ABB RAPID module: 3RHTCO_Mod1(Mod)_5000.mod

MODULE RHTCO1
    ! Code Developers: Linus Y L Ang and Zhang Zhiqian (IHPC/EM)
    ! Version Date/Time: 2024.12.02 / 16:41

    ! Get input coordinates.
    PERS num x_coords_rel{5000}:=[0.0, 0.2, 0.0, 0.1, 0.0, 0.2, 0.0, 0.1, 0.0, 0.2, 0.0, 0.0, -0.2, 0.0, -0.1, 0.0, 0.0, -0.2, 0.0, -0.1, 0.0, 0.0, -0.2, 0.0, -0.2, 0.0, 0.0, -0.1, 0.0, -0.2, 0.0, -0.1, -4.9, 0.0, 5.0, 0.0, 0.2, 0.0, 0.1, 0.0, 0.2, 0.0, 0.2, 0.0, 0.1, 0.0, 0.2, 0.0, 0.1, 0.0, 0.2, 0.0, 0.0, 0.0, -0.2, 0.0, -0.1, 0.0, -0.2, 0.0, -0.1, 0.0, 0.0, -0.2, 0.0, -0.2, 0.0, -0.1, 0.0, -0.2, 0.0, 0.0, -0.1, -4.9, 0.0, 4.9, 0.0, 0.1, 0.0, 0.2, 0.0, 0.1, 0.0, 0.2, 0.0, 0.2, 0.0, 0.1, 0.0, 0.2, 0.0, 0.1, 0.0, 0.2, 0.0, 0.0, -0.2, 0.0, -0.1, 0.0, -0.2, 0.0, -0.1, 0.0, 0.0, -0.2, 0.0, -0.2, 0.0, -0.1, 0.0, -0.2, 0.0, -0.1, -0.2, -4.7, 0.0, 4.7, 0.0, 0.2, 0.1, 0.0, 0.2, 0.1, 0.0, 0.2, 0.0, 0.2, 0.0, 0.1, 0.0, 0.2, 0.0, 0.1, 0.0, 0.2, 0.0, 0.2, -0.2, 0.0, -0.2, 0.0, -0.1, 0.0, 0.0, -0.2, 0.0, -0.1, 0.0, -0.2, 0.0, -0.2, 0.0, -0.1, 0.0, -0.2, 0.0, -0.1, -4.9, 0.0, 4.9, 0.0, 0.1, 0.2, 0.0, 0.0, 0.1, 0.0, 0.2, 0.0, 0.2, 0.0, 0.1, 0.0, 0.2, 0.0, 0.1, 0.0, 0.2, 0.0, 0.2, 0.0, 0.0, -0.2, 0.0, -0.2, 0.0, -0.1, -0.2, 0.0, -0.1, 0.0, -0.2, 0.0, -0.2, 0.0, -0.1, -0.2, 0.0, -0.1, 0.0, -0.2, -0.2, -0.1, -0.2, -0.2, -1.1, -0.1, -1.2, -0.1, -1.1, -0.2, -0.2, 0.0, 0.2, 0.0, 0.2, 1.1, 0.1, 1.2, 0.1, 1.1, 0.2, 0.2, 0.1, 0.2, 0.2, 0.0, 0.0, 0.1, 0.0, 0.2, 0.0, 0.0, 0.1, 0.0, 0.0, 0.2, 0.0, 0.0, 0.2, -0.2, -0.2, -0.1, -0.2, -1.0, -0.1, -1.0, -0.1, -1.2, -0.1, 0.0, 0.1, 1.2, 0.1, 1.0, 0.1, 1.0, 0.2, 0.1, 0.2, 0.2, 0.1, 0.0, 0.2, 0.1, 0.2, 0.2, 0.1, 0.2, 0.1, 0.2, 0.2, 0.1, 0.2, 0.0, -0.2, 0.0, -0.1, 0.0, -0.2, -0.2, -0.1, -0.2, -0.1, -0.2, -0.2, -0.1, -0.2, -0.1, -0.2, 0.0, 0.2, 0.1, 0.2, 0.1, 0.2, 0.2, 0.1, 0.2, 0.1, 0.8, 0.0, 0.2, 0.2, 0.1, 0.2, 0.1, 0.2, 0.2, 0.1, 0.2, 0.2, 0.1, 0.2, 0.1, 0.2, 0.2, 0.1, 0.2, 0.1, 0.0, -0.1, 0.0, -0.2, 0.0, -0.1, 0.0, -0.2, -0.2, -0.1, -0.2, -0.1, -0.2, -0.2, -0.1, -0.2, -0.2, -0.1, -0.2, -0.1, -0.2, -0.2, -0.1, -0.2, -0.1, -0.2, -0.2, -0.1, -0.7, -0.1, -0.7, -0.1, -0.2, -0.1, -0.2, -0.2, -0.8, 0.0, 0.2, 0.0, 0.0, 0.1, 0.0, 0.0, 0.0, 0.2, 0.0, 0.0, 0.2, 0.0, 0.0, 0.1, 0.0, -0.1, 0.0, -0.2, 0.0, 0.0, -0.2, 0.0, 0.0, -0.1, 0.0, 0.0, 0.0, -0.2, 0.0, 0.0, -0.1, 0.0, -0.2, -0.2, -0.1, -0.2, -0.1, -0.2, -0.2, -0.1, -0.2, -0.1, -0.2, -0.2, -0.1, -0.2, -0.1, -0.2, -0.2, -0.1, -0.2, -0.1, -3.27, -0.16, 3.43, -0.2, 0.0, 0.0, 0.0, -0.2, 0.0, 0.0, 0.0, -0.13, 0.0, 0.0, 0.0, -0.16, 0.0, 0.0, -0.16, -0.16, -0.17, -0.16, -0.16, -0.16, -0.16, -0.16, -0.16, -0.16, -0.16, -0.16, -0.16, -0.16, -0.16, -0.17, -0.16, -0.16, -0.16, -0.16, -0.16, -0.16, -0.16, -0.16, -0.16, -0.16, -0.16, -0.16, -0.17, -0.16, -0.16, -0.16, -0.16, -0.16, -0.16, -0.16, -0.16, -0.16, -0.16, -0.16, -0.16, -0.17, -0.16, -0.16, -0.16, -0.16, 0.16, 0.16, 0.16, 0.16, 0.17, 0.16, 0.16, 0.16, 0.16, 0.16, 0.16, 0.16, 0.16, 0.16, 0.16, 0.16, 0.16, 0.17, 0.16, 0.16, 0.16, 0.16, 0.16, 0.16, 0.0, -0.8, -4.34, 0.0, 4.18, 0.0, 0.16, 0.0, 0.0, 0.16, 0.0, 0.16, 0.0, 0.16, 0.0, 0.16, 0.0, 0.16, 0.0, 0.16, 0.0, 0.0, -0.16, -0.16, -0.16, -0.16, -0.16, -0.16, -0.16, -0.17, -0.16, -0.16, -0.16, -0.16, -0.16, -0.16, -0.16, -0.16, 0.0, 0.16, 0.16, 0.16, 0.16, 0.16, 0.16, 0.16, 0.16, 0.17, 0.16, 0.16, 0.16, 0.16, 0.16, 0.16, 0.16, 0.0, -0.16, 0.0, -0.16, 0.0, -0.16, 0.0, -0.16, 0.0, -0.16, 0.0, 0.64, 0.16, 0.0, 0.16, 0.16, 0.16, 0.16, 0.16, 0.17, 0.16, 0.16, 0.16, 0.16, 0.16, 0.16, 0.16, 0.16, 0.16, 0.16, 0.16, 0.16, 0.17, 0.16, 0.16, 0.29, 0.0, 0.0, 0.0, 0.2, 0.0, 0.0, 0.0, 0.2, 0.0, 0.0, 0.0, 0.1, 0.2, 0.1, 0.2, 0.2, 0.1, 0.2, 0.1, 0.2, 0.2, 0.1, 0.2, 0.1, 0.2, 0.2, 0.1, 0.2, 0.1, 0.2, 0.2, 0.0, 0.1, 0.2, 0.6, 0.2, 0.2, 0.1, 0.2, 0.1, 0.7, 0.1, 0.7, 0.1, 0.2, 0.2, 0.1, 0.2, 0.1, 0.0, 0.0, 0.0, -0.1, 0.0, 0.0, -0.2, 0.0, 0.0, -0.1, 0.0, 0.0, -0.2, 0.0, 0.0, 0.0, -0.2, 0.0, 0.0, -0.1, -0.2, -0.1, -0.2, -0.2, -0.1, -0.2, -0.1, -0.2, -0.2, -0.1, -0.2, -0.1, -0.2, -0.2, -0.1, -0.2, -0.2, 0.0, 0.2, 0.2, 0.1, 0.2, 0.2, 0.1, 0.2, 0.1, 0.2, 0.2, 0.1, 0.2, 0.1, 0.2, 0.2, 0.1, 0.2, 0.1, 0.4, 0.0, 0.0, 0.0, 0.1, 0.0, 0.0, 0.2, 0.0, 0.0, 0.1, 0.0, 0.0, 0.2, 0.0, 0.0, 0.2, 0.1, 0.2, 0.1, 0.2, 0.2, 0.1, 0.2, 0.2, 0.1, 0.2, 0.1, 0.2, 0.6, 0.0, 0.2, 0.2, 0.1, 0.2, 0.1, 0.2, 0.2, 0.1, 0.2, 0.1, 0.2, 0.2, 0.1, 0.2, 0.2, 0.1, 0.2, 0.1, 0.2, 0.2, 0.0, 0.0, 0.0, 0.1, 0.0, 0.0, 0.0, 0.2, 0.0, 0.0, 0.0, 0.1, 0.0, 0.0, 0.2, 0.0, 0.0, 0.0, 0.2, 0.0, 0.0, 0.0, 0.1, 0.0, 0.0, 0.0, -0.1, 0.0, -0.2, -0.2, -0.1, -0.2, -0.1, -0.2, -0.2, -0.1, -0.2, -0.1, -0.2, -0.2, -0.1, -0.2, -0.2, -0.1, -0.2, -0.1, -0.2, -0.2, -0.1, -0.2, -0.1, -0.2, 0.0, 0.2, 0.1, 0.2, 0.1, 0.2, 0.2, 0.1, 0.2, 0.1, 0.2, 0.2, 0.1, 0.2, 0.2, 0.1, 0.2, 0.1, 0.2, 0.2, 0.1, 0.2, 0.1, 0.2, 0.0, 0.2, 0.0, 0.1, 0.0, 0.2, 0.0, 0.0, 0.1, 0.0, 0.2, 0.0, 0.0, 0.2, 0.0, 0.1, 0.0, 0.2, 0.0, 0.0, 0.1, 0.0, 0.2, 0.0, 0.2, 0.0, 0.0, -0.2, -0.2, 0.0, -0.1, -0.2, 0.0, -0.1, -0.2, -0.2, 0.0, -0.1, -0.2, 0.0, -0.1, -0.2, 0.0, -0.2, -0.1, -0.2, 0.0, -0.1, -0.2, -0.2, -0.8, -0.1, -0.2, -0.2, 0.0, 0.2, 0.2, 0.1, 1.0, 0.5, 0.0, 0.1, 0.2, 0.2, 0.0, 0.1, 0.2, 0.0, 0.1, 0.2, 0.0, 0.2, 0.1, 0.2, 0.0, 0.1, 0.2, 0.0, 0.2, 0.1, -0.1, -0.2, 0.0, -0.2, 0.0, 0.0, -0.1, 0.0, -0.2, 0.0, -0.1, 0.0, 0.0, -0.2, 0.0, -0.2, 0.0, 0.0, -0.1, 0.0, -0.2, 0.0, -0.1, 0.0, 0.1, 0.0, 0.2, 0.1, 0.2, 0.2, 0.1, 0.2, 0.6, 0.2, 0.1, 0.2, 0.2, 0.1, 0.2, 0.2, 0.1, 0.2, 0.6, 0.2, 0.1, 0.2, 0.2, 0.1, 0.2, 0.1, 0.2, 0.2, 0.6, 0.0, -0.6, -0.2, -0.2, -0.1, -0.2, -0.1, -0.2, -0.2, -0.1, -0.2, -0.6, -0.2, -0.1, -0.2, -0.2, -0.1, -0.2, -0.2, -0.1, -0.2, -0.6, -0.2, -0.1, -0.2, -0.2, -0.1, -0.2, 0.0, 0.0, 0.0, -0.1, 0.0, 0.0, 0.0, -0.2, 0.0, 0.0, -0.2, 0.0, 0.0, 0.0, -0.1, 0.0, 0.0, 0.0, -0.2, 0.0, 0.0, 0.0, -0.1, 0.0, 0.8, 0.1, 1.1, 0.2, 1.0, 0.1, 0.0, -0.1, -1.0, -0.2, -1.1, -0.1, -0.8, -0.2, -0.2, -0.1, -0.2, -0.1, -0.2, -0.2, -0.1, -0.2, -0.2, -0.1, -0.2, -0.1, -0.2, -0.2, -0.1, -0.2, -0.1, -0.2, -0.2, -0.1, -0.2, 0.0, 0.2, 0.0, 0.1, 0.0, 0.2, 0.0, 0.0, 0.2, 0.1, 0.2, 0.1, 0.2, 0.2, 0.0, -0.2, -0.2, -0.1, -0.2, -0.1, -0.2, -0.2, -0.1, -0.2, -0.1, -0.2, -0.2, -0.1, -0.2, -0.1, -0.2, -0.2, -0.1, -0.2, -0.2, -0.1, -0.2, -0.1, -0.2, -0.2, -0.1, -0.2, 0.0, 0.2, 0.0, 0.1, 0.0, 0.2, 0.2, 0.1, 0.2, 0.8, 0.2, 0.8, 0.1, 0.8, 0.2, 0.0, -0.2, -0.8, -0.1, -0.8, -0.2, -0.8, -0.2, -0.6, -0.2, -0.1, -0.2, -0.2, -0.1, -0.2, -0.1, -0.2, -0.2, -0.1, -0.2, -0.1, 0.0, 0.0, -0.2, 0.0, 0.0, -0.2, 0.0, 0.0, -0.1, 0.0, -0.2, 0.0, 0.0, -0.1, 0.0, 0.0, 0.1, 0.0, 0.2, 0.0, 0.1, 0.2, 0.0, 0.2, 0.0, 0.1, 0.0, 0.2, 0.0, 0.1, 0.2, 0.0, 0.2, 0.0, 0.1, 4.7, 0.0, -4.5, -0.2, -0.1, 0.0, -0.2, 0.0, -0.2, 0.0, -0.1, 0.0, -0.2, 0.0, -0.1, 0.0, -0.2, 0.0, -0.2, 0.0, 0.0, -0.1, 0.0, -0.2, 0.2, 0.0, 0.1, 0.0, 0.2, 0.0, 0.2, 0.0, 0.1, 0.0, 0.2, 0.0, 0.1, 0.0, 0.0, 0.2, 0.0, 0.2, 0.1, 4.5, 0.0, -4.5, -0.1, 0.0, -0.2, 0.0, -0.2, 0.0, -0.1, 0.0, -0.2, 0.0, -0.1, 0.0, -0.2, 0.0, -0.2, -0.1, 0.0, -0.2, 0.0, 0.0, 0.0, 0.2, 0.0, 0.1, 0.0, 0.2, 0.0, 0.2, 0.0, 0.1, 0.0, 0.0, 0.2, 0.0, 0.1, 0.0, 0.2, 0.0, 0.2, 0.1, 4.7, 0.0, -4.8, -0.2, 0.0, -0.2, 0.0, -0.1, 0.0, -0.2, 0.0, -0.1, 0.0, -0.2, 0.0, -0.2, 0.0, -0.1, 0.0, -0.2, 0.0, 0.2, 0.0, 0.0, 0.1, 0.0, 0.2, 0.0, 0.2, 0.0, 0.1, 0.0, 0.0, 0.2, 0.0, 0.1, 0.0, 0.2, 0.0, 0.2, 0.1, 4.7, 0.0, -4.7, -0.1, -0.2, 0.0, -0.2, 0.0, -0.1, 0.0, -0.2, 0.0, -0.1, 0.0, -0.2, 0.0, -0.2, 0.0, -0.1, 0.0, 0.0, 0.0, 0.1, 0.0, 0.2, 0.0, 0.0, 0.2, 0.0, 0.1, 0.0, 0.0, 0.2, 0.0, 0.1, 0.0, 0.0, 0.2, 0.0, 0.2, 0.1, 4.7, 0.0, -4.8, -0.2, 0.0, -0.2, 0.0, -0.1, 0.0, -0.2, 0.0, -0.1, -0.2, 0.0, -0.2, 0.0, -0.1, 0.1, 0.0, 0.0, 0.2, 0.0, 0.0, 0.2, 0.0, 0.0, 0.1, 0.0, 0.0, 0.2, 0.0, 0.0, 0.1, 0.0, 0.0, -0.1, 0.0, 0.0, -0.2, 0.0, 0.0, -0.1, 0.0, 0.0, -0.2, 0.0, 0.0, -0.2, 0.0, 0.0, -0.1, 0.0, -0.2, -5.78, -0.16, 0.0, 0.16, 0.98, 0.2, 1.7, 0.2, 1.7, 0.2, 0.0, -0.2, -1.7, -0.2, -1.7, -0.2, -0.98, -0.16, 0.0, 0.16, 0.17, 0.16, 0.16, 0.16, 0.13, 0.2, 0.2, 0.1, 0.2, 0.1, 0.2, 0.2, 0.1, 0.2, 0.1, 0.0, -0.1, -0.2, -0.1, -0.2, -0.2, -0.1, -0.2, -0.1, -0.2, -0.2, -0.13, -0.16, -0.16, -0.16, -0.17, -0.16, -0.16, -0.16, -0.16, -0.64, 0.0, -0.64, 0.0, -0.17, -0.16, 0.0, -0.16, -0.16, 0.0, -0.16, 0.0, -0.16, 0.0, -0.16, 0.0, 0.0, -0.16, 0.0, -0.16, 0.0, 0.0, -0.16, 0.0, 0.16, 0.16, 0.16, 0.16, 0.16, 0.16, 0.16, 0.16, 0.16, 0.17, 0.16, 0.16, 0.16, 0.16, 0.16, 0.16, 0.16, 0.16, 0.16, 0.16, 0.16, 0.16, 0.17, 0.16, 0.16, 0.16, 0.13, 0.2, 0.2, 0.1, 0.2, 0.1, 0.2, 0.2, 0.0, -0.2, -0.2, -0.1, -0.2, -0.1, -0.2, -0.2, -0.13, -0.16, -0.16, -0.16, -0.17, -0.16, -0.16, -0.16, -0.16, -0.16, -0.16, -0.16, -0.16, -0.16, -0.16, -0.16, -0.16, -0.17, -0.16, -0.16, -0.16, -0.16, -0.16, -0.16, -0.16, -0.16, -0.16, -0.16, 0.0, -0.16, 0.0, 0.16, 0.0, 0.16, 0.0, 0.0, 0.0, 0.16, 0.0, 0.0, 0.16, 0.0, 0.16, 0.0, 0.0, 0.16, 0.0, 0.16, 0.16, 0.16, 0.16, 0.0, 0.16, 0.17, 0.0, 0.64, 0.0, 0.96, 0.16, 0.65, 0.16, 0.13, 0.2, 0.2, 0.1, 0.2, 0.1, 0.2, 0.2, 0.1, 0.2, 0.1, 0.2, 0.2, 0.1, 0.0, 0.2, 0.1, 0.0, 0.2, 0.0, 0.0, 0.2, 0.0, 0.0, 0.1, 0.0, 0.0, 0.2, 0.0, 0.0, 0.1, 0.0, 0.0, 0.2, 0.0, 0.2, 0.0, 0.0, 0.1, 0.0, 0.0, 0.2, 0.0, 0.0, 0.1, 0.0, 0.0, 0.2, 0.2, -0.2, 0.0, 0.0, -0.2, 0.0, 0.0, -0.1, 0.0, 0.0, -0.2, 0.0, 0.0, -0.1, 0.0, -0.2, 0.0, 0.0, -0.2, 0.0, 0.0, -0.1, 0.0, 0.0, -0.2, 0.0, 0.0, -0.1, 0.0, 0.0, -0.2, 0.0, -0.2, 0.0, 0.2, 0.2, 0.1, 0.2, 0.1, 0.2, 0.2, 0.1, 0.2, 0.6, 0.2, 2.4, 0.0, 0.2, 0.6, 0.2, 0.6, 0.2, 0.1, 0.2, 0.2, 0.1, 0.2, 0.1, 0.0, 0.0, -0.1, 0.0, -0.2, 0.0, 0.0, -0.1, 0.0, -0.2, 0.0, -0.2, 0.0, 0.0, -0.1, 0.0, -0.2, 0.0, 0.0, -0.2, 0.0, -0.1, 0.0, 0.0, -0.2, 0.0, -0.1, 0.0, -0.2, 0.0, 0.0, -0.2, 0.0, 0.2, 0.0, 0.2, 0.0, 0.0, 0.1, 0.0, 0.2, 0.0, 0.1, 0.0, 0.0, 0.2, 0.0, 0.2, 0.0, 0.0, 0.1, 0.0, 0.2, 0.0, 0.0, 0.2, 0.0, 0.1, 0.0, 0.2, 0.0, 0.0, 0.1, 0.0, 0.2, 0.2, 0.1, 0.0, 0.2, 0.1, 0.2, 0.2, 0.1, 0.2, 0.1, 0.2, 0.2, 0.1, 0.2, 0.1, 0.2, 0.2, 0.1, 1.3, 0.0, 0.7, 0.0, 0.1, 0.0, 0.2, 0.1, 0.0, 0.2, 0.0, 0.2, 0.0, -0.2, -0.2, -0.1, -0.2, -0.1, -0.2, -0.2, -0.1, -0.2, -0.1, -0.2, -0.2, -0.1, -0.2, -0.1, -0.2, -0.2, -0.1, -0.2, -0.2, -0.1, -0.2, -0.1, -0.2, -0.2, -0.1, -0.2, -0.1, -0.2, -0.2, 0.0, 0.2, 0.2, 0.1, 0.2, 0.1, 0.2, 0.2, 0.1, 0.2, 0.1, 0.2, 0.2, 0.1, 0.2, 0.2, 0.1, 0.2, 0.1, 0.2, 0.2, 0.1, 0.2, 0.1, 0.2, 0.2, 0.1, 0.2, 0.1, 0.2, 0.2, 0.1, 0.0, 0.2, 0.0, 0.0, 0.1, 0.0, 0.0, 0.2, 0.0, 0.0, 0.2, 0.0, 0.1, 0.0, 0.2, 0.0, -0.2, 0.0, -0.1, 0.0, -0.2, 0.0, 0.0, -0.2, -0.1, -0.2, -0.1, -0.2, -0.2, -0.1, -0.2, -0.1, -0.2, -0.2, -0.1, -0.2, -0.1, -0.2, -0.2, -0.1, -0.2, -0.1, -0.2, -0.2, -0.1, -0.2, -0.2, -0.1, -0.2, -0.1, -0.2, -0.2, -0.1, -0.2, -0.1, -0.2, -0.2, -0.1, 0.0, 0.1, 0.2, 0.2, 0.1, 0.2, 0.1, 0.2, 0.2, 0.1, 0.2, 0.1, 0.2, 0.2, 0.1, 0.2, 0.2, 0.1, 0.2, 0.1, 0.2, 0.2, 0.1, 0.2, 0.1, 0.2, 0.2, 0.1, 0.2, 0.1, 0.2, 0.2, 0.1, 0.2, 0.1, -0.1, 0.0, 0.0, -0.2, 0.0, -0.1, 0.0, -0.2, 0.0, -0.2, 0.0, -0.1, -0.2, 0.0, -0.1, 0.0, -0.2, -0.2, -0.1, 0.0, -1.1, -0.2, -0.7, 0.0, 0.0, -0.1, -0.2, -0.1, -0.2, -0.2, -0.1, -0.2, -0.1, -0.2, -0.2, -0.1, -0.2, -0.1, -0.2, -0.2, -0.1, 0.0, -0.2, 0.0, 0.0, -0.1, 0.0, 0.0, 0.0, -0.2, 0.0, 0.0, 0.0, -0.2, 0.0, 0.0, 0.0, -0.1, 0.0, 0.0, -0.2, 0.0, 0.0, 0.0, -0.2, 0.0, 0.0, 0.0, 0.2, 0.0, 0.0, 0.2, 0.0, 0.0, 0.0, 0.1, 0.0, 0.0, 0.0, 0.2, 0.0, 0.0, 0.0, 0.2, 0.0, 0.0, 0.1, 0.0, -0.1, -0.2, -0.2, -0.1, -0.2, -0.2, -0.1, -0.2, -0.1, -0.2, -0.2, -0.1, -0.2, -0.1, -0.2, -0.2, -0.1, 0.0, 0.1, 0.2, 0.2, 0.1, 0.2, 0.1, 0.2, 0.2, 0.1, 0.2, 0.1, 0.2, 0.2, 0.1, 0.2, 0.2, 0.6, 0.0, 0.2, 0.1, 0.2, 0.1, 0.2, 0.2, 0.1, 0.2, 0.1, 0.2, 0.2, 0.1, 0.2, 0.1, 0.0, -0.1, -5.6, -0.2, 0.0, -0.2, 0.0, -0.1, -0.2, 0.0, -0.1, 0.0, -0.2, -0.2, 0.0, 0.2, 0.0, 0.2, 0.0, 0.0, 1.4, 0.0, 0.2, 0.0, 0.1, 0.1, 0.1, 0.1, 0.1, 0.1, 0.2, 0.0, 0.1, 0.2, 0.0, 0.1, 0.2, 0.1, 0.1, 0.1, 0.0, 0.2, 0.0, 0.2, 0.1, 0.1, 0.1, 0.0, 0.1, 0.0, 0.2, 0.2, 0.1, 0.0, 0.2, 0.1, 0.0, 0.2, 0.2, 0.1, 0.0, 0.2, 0.1, 0.0, 0.2, 0.1, 0.0, -0.1, -4.7, -0.1, 0.0, -0.1, 0.0, -0.1, -0.1, 0.0, -0.1, -0.1, 0.0, -0.1, 0.0, -0.1, 0.0, -0.1, -0.1, 0.0, 0.1, 0.0, 0.1, 0.0, 0.0, 0.0, 0.0, 0.1, 0.0, 0.0, 0.0, 1.4, 0.0, 0.1, 0.0, 0.2, 0.0, 0.2, 0.0, 0.1, 0.2, 0.1, 0.0, 0.2, 0.1, 0.1, 0.1, 0.1, 0.1, 0.1, 0.1, 0.1, 0.1, 0.1, 0.0, 0.1, 0.0, 0.2, 0.2, 0.0, 0.1, 0.2, 0.1, 0.0, 0.2, 0.2, 0.0, 0.1, 0.0, -0.1, -3.6, -0.1, -0.2, 0.0, -0.1, -0.1, 0.0, -0.1, 0.0, -0.1, 0.0, -0.1, 0.0, 0.0, 0.0, 0.1, 0.0, 0.0, 0.0, 0.1, 0.0, 1.2, 0.0, 0.1, 0.1, 0.0, 0.2, 0.1, 0.0, 0.2, 0.1, 0.1, 0.1, 0.1, 0.1, 0.2, 0.0, 0.1, 0.1, 0.1, 0.1, 0.0, 0.1, 0.1, 0.2, 0.0, 0.1, 0.2, 0.0, 0.0, 0.0, -2.9, 0.0, -0.2, 0.0, -0.1, 0.0, -0.1, 0.0, 0.0, 0.1, 0.0, 1.4, 0.0, 0.1, 0.1, 0.1, 0.2, 0.0, 0.2, 0.1, 0.0, 0.2, 0.1, 0.0, 0.0, 0.1, 0.0, 0.0, -0.1, -1.9, -0.1, 1.1, 0.6, 0.1, 0.0, -0.1, 0.0, 0.0, 0.0, -0.1, -0.2, 0.0, -0.2, -1.5, 0.0, 0.0, 0.1, 0.0, 0.1, 0.0, 2.5, 0.0, 0.0, 0.0, 0.0, -0.2, -0.1, -0.1, 0.0, 0.0, -0.1, -0.2, 0.0, -0.1, -0.2, -0.1, -0.1, -0.1, -0.1, -0.1, -0.2, 0.0, -0.1, 0.0, -1.4, 0.0, 0.0, 0.0, -0.1, 0.0, 0.0, 0.0, 0.1, 0.1, 0.0, 0.1, 0.1, 0.0, 0.1, 0.2, 3.0, 0.2, 0.0, -0.1, -0.1, -0.1, -0.2, -0.1, 0.0, -0.2, -0.1, -0.1, 0.0, -0.1, -0.1, -0.1, -0.1, 0.0, -0.2, -1.0, 0.0, -0.1, -0.2, 0.0, -0.2, 0.0, -1.2, 0.0, 0.0, 0.0, -0.1, 0.0, 0.0, 0.0, -0.1, 0.0, 0.0, 0.0, 0.0, 0.1, 0.1, 0.0, 0.1, 0.0, 0.1, 0.1, 0.0, 0.1, 0.0, 0.1, 0.1, 4.2, 0.1, 0.0, -0.1, 0.0, -0.2, 0.0, -0.1, -0.2, -0.2, 0.0, -0.1, -0.2, 0.0, -0.1, -0.2, -0.2, 0.0, -0.1, 0.0, -0.1, -0.1, -0.1, -0.1, -0.1, -0.2, 0.0, -0.1, -0.1, -0.1, -0.2, -0.1, 0.0, -0.2, -0.1, 0.0, -0.2, -0.1, -0.1, -0.1, 0.0, -0.2, -0.1, 0.0, 0.0, -1.4, 0.0, 0.0, 0.0, 0.0, -0.1, 0.0, 0.0, 0.0, 0.0, 0.0, -0.1, 0.0, -0.1, 0.0, 0.1, 0.0, 0.1, 0.0, 0.1, 0.1, 0.0, 0.1, 0.0, 0.0, 0.2, 0.0, 0.1, 0.1, 0.0, 0.1, 0.0, 0.0, 0.2, 5.1, 0.1, 0.0, -0.1, 0.0, -0.1, -0.2, -0.2, 0.0, -0.1, -0.2, 0.0, -0.1, -0.2, -0.2, 0.0, -0.1, -0.2, 0.0, -0.1, -0.2, -0.2, 0.0, 0.0, -0.1, -0.2, 0.0, -0.1, -0.2, 0.0, -0.2, -0.1, 0.0, -0.2, 0.0, -0.2, -0.1, 0.0, -0.2, -0.1, 0.0, -0.2, -0.2, 0.0, -0.1, -0.2, 0.0, -0.1, 0.0, -0.2, -0.2, 0.0, -1.2, -1.5, 0.0, -1.6, 0.0, 0.0, 0.2, 0.0, 0.0, 0.1, 0.0, 0.0, 0.2, 0.0, 0.0, 0.1, 0.0, 0.0, 0.2, 0.0, 0.2, 0.0, 0.0, 0.1, 0.0, 0.2, 0.1, 0.2, 0.2, 0.1, 0.2, 0.2, 0.1, 0.2, 0.1, 0.2, 0.2, 0.1, 0.2, 0.1, 0.2, 0.2, 0.1, 0.2, 0.1, 0.2, 0.2, 0.1, 0.2, 0.1, 0.0, 0.2, 0.0, 0.1, 0.1, 0.0, 0.0, 0.1, 0.0, 0.0, 0.1, 0.1, 0.0, 0.0, 0.1, 0.0, 0.0, 0.1, 0.0, 0.1, -0.2, -0.1, -0.2, -0.1, -0.2, -0.2, -0.1, -0.2, -0.1, -0.2, -0.2, -0.1, -0.2, -0.1, -0.2, -0.2, -0.1, -0.2, -0.9, -0.1, -0.1, -1.3, 0.0, 0.0, 0.1, 0.0, 0.1, 0.1, 0.0, 0.0, 0.1, 0.1, 0.0, 0.1, 0.0, 0.1, 0.1, 0.2, 0.1, 0.2, 0.2, 0.1, 0.2, 0.1, 0.2, 0.2, 0.1, 0.2, 0.1, 0.2, 0.2, 0.1, 0.2, 0.1, 0.2, 0.0, 0.5, 0.0, 0.0, 0.0, 0.0, 0.1, 0.0, 0.0, 0.1, 0.0, 0.0, 0.1, 0.0, 0.0, 0.0, -0.1, -0.1, -0.1, 0.0, -0.2, -0.1, -0.1, -0.1, -0.2, 0.0, -0.1, -0.2, 0.0, -0.1, -0.1, -0.1, -0.2, 0.0, -0.1, -0.6, -0.1, 0.0, 0.0, -0.1, -0.1, -0.9, -0.1, 0.1, 0.0, 0.0, 0.1, 0.0, 0.1, 0.0, 0.0, 0.1, 0.0, 0.2, 0.0, 0.2, 0.1, 0.0, 0.2, 0.1, 0.2, 0.2, 0.1, 0.2, 0.1, 0.2, 0.2, 0.1, 0.0, 0.5, 0.0, 0.0, 0.1, -0.1, -0.2, -0.1, -0.2, -0.1, -0.2, -0.1, -0.1, 0.0, -0.1, -0.1, -0.1, 0.0, -0.1, 0.0, -0.1, -0.7, 0.0, 0.1, 0.2, 0.1, 0.2, 0.2, 0.1, 0.2, 0.1, 0.2, -0.3, -0.2, -0.1, 0.1, 0.0, 0.2, 0.1, 0.0, 0.2, 0.1, 0.1, 0.0, 0.0, 0.0, -0.2, -0.2, -0.1, -0.2, -0.1, -0.2, -0.2, -0.1, -0.2, -0.1, 0.0, -0.2, 0.0, -0.1, 0.0, -0.1, 0.0, 0.0, 0.0, 0.8, 0.1, 0.1, 0.0, 0.1, 0.1, 0.0, 0.1, 0.1, 0.1, 0.1, 0.1, 0.1, 0.2, 0.0, 0.1, 0.2, 0.1, 0.0, 0.2, 0.1, 0.1, 0.1, 0.1, 0.0, 0.0, 0.0, -0.1, 0.0, 0.0, -0.1, 0.0, -0.4, 0.0, -0.1, -0.1, -0.1, -0.1, -0.2, -0.2, -0.1, -0.2, -0.1, -0.2, -0.2, -0.1, -0.1, -0.1, -0.1, -0.1, -0.1, -0.2, -0.1, 0.0, -0.1, 0.0, -0.1, 0.0, 0.0, -0.1, -0.1, 0.0, 0.0, -0.1, 0.0, 0.0, -0.1, 0.0, -0.1, 0.0, 0.0, 1.2, 0.1, 0.0, 0.1, 0.1, 0.0, 0.6, 0.2, 0.1, 0.1, 0.1, 0.2, 0.0, 0.1, 0.1, 0.1, 0.1, 0.1, 0.1, 0.2, 0.0, 0.1, 0.2, 0.1, 0.0, 0.2, 0.0, 0.2, 0.0, 0.1, 0.1, -0.1, 0.0, 0.0, -0.1, 0.0, 0.0, -0.1, 0.0, -0.1, 0.0, 0.0, -0.1, 0.0, 0.0, -0.5, 0.0, -0.1, -0.1, -0.2, 0.0, -0.1, -0.2, -0.1, 0.0, -0.2, -0.2, -0.1, -0.2, -0.1, -0.2, -0.2, 0.0, -0.1, -0.2, -0.1, 0.0, -0.2, -0.1, -0.1, -0.1, -0.1, -0.1, -0.2, -0.1, 0.0, 0.0, -0.1, -0.1, 0.0, -0.1, 0.0, -0.1, -0.1, 0.0, 0.0, -0.1, -0.1, 0.0, -0.1, 0.0, 0.0, -0.1, 1.4, 0.1, 0.0, 0.1, 1.2, 0.2, 0.1, 0.0, 0.2, 0.1, 0.1, 0.1, 0.1, 0.1, 0.1, 0.0, 0.2, 0.1, 0.1, 0.1, 0.1, 0.1, 0.1, 0.1, 0.1, 0.2, 0.0, 0.1, 0.2, 0.0, 0.1, 0.1, 0.1, 0.2, 0.0, 0.1, 0.1, -0.1, 0.0, -0.1, 0.0, 0.0, -0.1, -0.1, 0.0, 0.0, 0.0, -0.1, -0.1, 0.0, 0.0, -0.1, 0.0, 0.0, -0.1, -0.1, 0.0, 0.0, 0.2, 0.0, 0.0, 0.0, 0.1, 0.2, 0.2, 0.1, 0.2, 0.2, 0.1, 0.2, 0.0, 0.0, 1.3, 0.0, 0.1, 0.2, 0.1, 0.2, 0.2, 0.1, 0.2, 0.1, 0.2, 0.2, 0.1, 0.2, 0.2, 0.1, 0.2, 0.1, 0.2, 0.2, 0.1, 0.2, 0.1, 0.2, 0.2, 0.1, 0.2, 0.0, 0.0, -0.1, -0.1, -0.1, 0.0, -0.1, -0.1, -0.2, -0.1, 0.0, -0.1, -0.1, -0.1, -0.2, -0.1, -0.1, -0.8, -0.1, -0.2, -0.6, -0.2, -0.2, -0.1, -0.2, -0.1, -0.2, -0.2, -0.1, -0.2, 0.0, -0.1, -0.1, 0.0, -0.1, 0.0, 0.0, -0.1, -0.1, 0.0, 0.0, 0.0, -0.1, 0.0, 0.0, -0.1, -0.1, 0.0, -0.1, 0.0, 0.0, -0.1, 0.0, -0.1, 0.0, 0.0, 0.2, 0.1, 0.2, 0.1, 0.2, 0.0, 1.4, 0.0, 0.2, 0.2, 0.0, 0.1, 0.2, 0.1, 0.2, 0.0, 0.2, 0.1, 0.2, 0.0, 0.2, 0.1, 0.2, 0.1, 0.0, 0.2, 0.2, 0.1, 0.0, 0.1, -0.1, 0.0, -0.1, 0.0, -0.1, -0.1, 0.0, -0.1, -0.1, 0.0, -0.1, 0.0, -0.1, -0.1, -0.1, 0.0, -0.1, -0.1, -0.5, -0.2, 0.0, -0.1, -0.1, -0.1, -0.3, -0.2, -0.1, -0.2, 0.0, -0.1, -0.2, 0.0, -0.1, -0.1, 0.0, 0.0, 0.0, 0.0, -0.1, 0.0, 0.0, -0.1, 0.0, -0.1, 0.0, 0.0, 0.0, -0.1, 0.0, 0.0, -0.1, 0.0, -0.1, 0.0, 0.0, 0.0, 0.0, 0.0, 0.2, 0.1, 0.0, 1.3, 0.0, 0.2, 0.1, 0.2, 0.1, 0.2, 0.2, 0.1, 0.2, 0.2, 0.0, 0.0, -0.1, -0.1, -0.1, -0.1, 0.0, -0.1, 0.0, -0.1, -0.1, -0.1, -0.1, 0.0, -0.1, -0.1, -0.1, -0.1, 0.0, -0.2, 0.0, -0.2, -0.1, 0.0, -0.1, 0.0, -0.1, 0.0, 0.0, -0.1, 0.0, -0.1, 0.0, 0.0, -0.1, 0.0, 1.0, 0.0, -0.5, 0.0, 0.0, 0.1, 0.0, 0.0, 0.0, 0.1, 0.1, 0.1, 0.1, 0.1, 0.0, 0.2, 0.0, 0.1, 0.0, 0.1, 0.1, 0.1, 0.1, 0.0, 0.0, -0.2, -0.2, 0.0, -0.1, -0.2, -0.1, 0.0, -1.5, 0.0, 0.0, 0.0, 0.1, 0.0, 0.0, 0.1, 0.0, 0.1, 0.0, 0.0, 0.0, 0.1, 0.0, 0.1, 0.0, 0.0, 0.0, 0.1, 0.0, 0.1, 0.0, 0.0, 0.1, 0.1, 0.1, 0.1, 0.1, 0.1, 0.1, 0.1, 0.1, 0.0, 0.2, 0.0, 0.1, 0.4, 0.1, 0.1, 0.1, 0.0, 0.1, 0.1, 0.0, 0.1, 0.0, 0.1, 0.1, 0.0, 0.1, 0.0, 0.1, -0.1, -0.1, 0.0, -0.2, -0.1, -0.2, -0.1, -0.1, -0.1, -0.2, -0.1, -0.1, -0.1, -0.2, -0.1, 0.0, -0.2, -0.2, 0.0, -1.4, 0.0, -0.1, -0.1, -0.1, -0.1, 0.0, 0.0, 0.1, 0.0, 0.0, 0.1, 0.0, 0.0, 0.1, 0.0, 0.1, 0.0, 0.0, 0.1, 0.0, 0.1, 0.0, 0.1, 0.0, 0.0, 0.1, 0.0, 0.1, 0.0, 0.1, 0.0, 0.2, 0.2, 0.1, 0.0, 0.2, 0.1, 0.0, 0.2, 0.5, 0.1, 0.1, 0.1, 0.2, 0.0, 0.6, 0.1, 0.1, 0.0, 0.1, 0.1, 0.1, 0.0, 0.1, 0.1, 0.0, 0.1, 0.0, 0.1, 0.1, 0.0, 0.1, 0.0, 0.1, 0.0, 0.1, 0.0, 0.0, 0.0, -0.2, -0.1, -0.2, 0.0, -0.1, -0.2, -0.2, -0.1, -0.2, -0.1, -0.2, 0.0, -0.2, -0.1, -0.2, 0.0, -0.2, -0.1, -0.2, -0.1, -0.2, -0.2, -0.1, 0.0, 0.0, -1.4, -0.2, -0.2, -0.1, 0.0, -0.2, -0.1, -0.1, -0.1, -0.1, 0.0, 0.1, 0.0, 0.0, 0.1, 0.0, 0.0, 0.1, 0.1, 0.0, 0.0, 0.1, 0.1, 0.0, 0.0, 0.1, 0.0, 0.0, 0.0, 0.1, 0.1, 0.0, 0.0, 0.1, 0.0, 0.1, 0.1, 0.0, 0.2, 0.1, 0.2, 0.1, 0.2, 0.1, 0.1, 0.1, 0.2, 0.1, 0.2, 0.1, 0.1, 0.1, 0.1, 0.1, 0.5, 0.1, 0.1, 0.1, 0.3, 0.6, 0.1, 0.0, 0.1, 0.3, 0.0, 0.1, 0.1, 0.0, 0.0, 0.1, 0.1, 0.1, 0.0, 0.0, 0.1, 0.1, 0.0, 0.1, 0.0, 0.1, 0.1, 0.0, 0.0, 0.1, 0.1, -0.2, -0.2, -0.1, -0.2, -0.1, -0.2, -0.2, -0.1, -0.2, -0.1, -0.2, -0.2, -0.1, -0.2, -0.1, -0.2, -0.2, -0.1, -0.2, -0.2, -0.1, -0.2, -0.1, -0.2, -0.2, -0.1, -0.2, -0.1, -0.2, -0.2, -0.8, 0.0, -0.1, 0.0, 0.0, 1.3, 0.0, 0.1, 0.2, 0.1, 0.2, 0.2, 0.1, 0.2, 0.1, 0.2, 0.2, 0.1, 0.2, 0.2, 0.1, 0.2, 0.1, 0.2, 0.2, 0.1, 0.2, 0.1, 0.2, 0.2, 0.1, 0.2, 0.1, 0.0, 0.2, 0.0, 0.1, 0.1, 0.0, 0.0, 0.1, 0.0, 0.0, 0.0, 0.1, 0.1, 0.0, 0.0, 0.1, 0.0, 0.0, -0.1, 0.0, 0.0, -0.1, -0.1, 0.0, 0.0, 0.0, -0.1, -0.2, -0.2, -0.1, -0.2, -0.1, -0.2, -0.2, -0.1, -0.2, -0.1, -0.2, -0.2, -0.1, -0.2, -0.1, -0.2, -0.2, -0.1, -0.2, -0.2, -0.1, -0.2, -0.1, -0.2, -0.2, -0.1, -0.2, -0.1, -0.2, -0.2, -0.1, -0.2, 0.0, 0.0, 1.3, 0.0, 0.0, 0.2, 0.1, 0.0, 0.2, 0.1, 0.1, 0.1, 0.2, 0.1, 0.0, 0.2, 0.2, 0.0, 0.1, 0.2, 0.0, 0.1, 0.2, 0.2, 0.0, 0.1, 0.2, 0.0, 0.1, 0.2, 0.0, 0.2, 0.1, 0.0, 0.1, 0.0, 0.1, 0.0, 0.0, 0.0, 0.1, 0.0, 0.0, 0.0, 0.1, 0.0, 0.0, 0.0, 0.0, -0.1, 0.0, 0.0, 0.0, -0.1, -0.2, -0.1, 0.0, -0.2, -0.2, -0.1, -0.1, -0.1, -0.1, -0.2, -0.1, -0.1, -0.1, -0.2, -0.1, 0.0, -0.2, -0.2, -0.1, -0.1, -0.1, -0.2, -0.1, -0.1, -0.1, -0.1, -0.2, -0.1, -0.1, -0.1, -0.2, -0.1, 0.0, 0.0, 0.0, 1.2, 0.0, 0.2, 0.2, 0.1, 0.2, 0.2, 0.1, 0.2, 0.1, 0.2, 0.2, 0.1, 0.2, 0.1, 0.0, 0.1, 0.0, 0.1, 0.0, 0.0, 0.0, 0.1, -0.1, 0.0, 0.0, 0.0, -0.2, -0.1, -0.2, -0.1, -0.2, -0.2, -0.1, -0.2, -0.1, -0.2, -0.2, -0.1, -0.2, -0.2, 0.0, 1.1, 0.0, 0.1, 0.1, 0.2, 0.0, 0.2, 0.0, 0.0, 0.0, -0.1, -0.1, -0.2, -0.1, -0.5, 0.2, 0.1, 0.1, 0.1, 0.1, 0.2, 0.1, 0.1, 0.1, 0.2, 0.0, 0.0, 0.0, 0.0, 0.0, 0.0, 0.0, 0.0, -0.2, 0.0, -0.1, -0.2, -0.1, -0.1, -0.1, -0.1, -0.1, -0.1, -0.2, 0.0, 0.0, -1.5, 0.0, 0.1, 0.1, 0.2, 0.1, 0.1, 0.1, 0.1, 0.2, 0.1, 0.1, 0.1, 0.2, 0.2, 0.0, 0.1, 0.2, 0.1, 0.1, 0.1, 0.2, 0.1, 0.2, 0.0, 0.1, 0.2, 0.2, 0.1, 0.0, 0.0, 0.0, 0.0, 0.0, 0.1, -0.1, 0.0, 0.0, 0.0, 0.0, -0.1, 0.0, 0.0, 0.0, -0.2, 0.0, -0.2, 0.0, -0.1, -0.2, -0.1, 0.0, -0.2, -0.2, 0.0, -0.1, -0.2, -0.1, 0.0, -0.2, -0.1, -0.1, -0.1, -0.2, -0.1, -0.1, -0.1, -0.1, -0.1, 0.0, -1.3, 0.0, 0.2, 0.2, 0.1, 0.2, 0.1, 0.0, 0.2, 0.2, 0.1, 0.0, 0.2, 0.1, 0.2, 0.2, 0.1, 0.2, 0.1, 0.1, 0.1, 0.2, 0.1, 0.0, 0.2, 0.2, 0.1, 0.2, 0.1, 0.2, 0.1, 0.1, 0.1, 0.2, 0.1, 0.0, 0.2, 0.0, 0.0, 0.1, 0.1, 0.0, 0.0, 0.0, 0.1, -0.1, 0.0, 0.0, 0.0, -0.1, -0.1, 0.0, 0.0, 0.0, 0.0, -0.1, 0.0, -0.1, 0.0, -0.1, 0.0, 0.0, -0.1, -0.1, -0.1, -0.2, 0.0, -0.2, -0.1, -0.1, -0.1, -0.1, -0.1, -0.1, -0.2, -0.1, -0.1, -0.1, -0.1, -0.1, -0.1, -0.2, 0.0, -0.1, -0.2, -0.2, 0.0, -0.1, -0.2, 0.0, -0.1, -0.2, -0.1, -0.1, 0.0, -1.4, 0.0, 0.2, 0.1, 0.2, 0.1, 0.2, 0.2, 0.1, 0.2, 0.1, 0.2, 0.2, 0.1, 0.2, 0.1, 0.2, 0.2, 0.1, 0.2, 0.2, 0.1, 0.2, 0.1, 0.2, 0.2, 0.1, 0.2, 0.1, 0.2, 0.2, 0.1, 0.2, 0.1, 0.2, 0.2, 0.1, 0.2, 0.0, 0.1, 0.0, 0.0, 0.0, 0.1, 0.1, 0.0, 0.0, 0.0, 0.1, 0.1, -0.1, -0.1, 0.0, 0.0, 0.0, -0.1, -0.1, 0.0, 0.0, 0.0, -0.1, 0.0, -0.1, 0.0, -0.1, 0.0, -0.1, 0.0, -0.2, 0.0, -0.2, 0.0, -0.1, -0.2, -0.1, 0.0, -0.2, -0.2, -0.1, -0.2, -0.1, 0.0, -0.2, -0.1, -0.1, -0.1, -0.2, -0.1, -0.2, -0.1, -0.1, -0.1, -0.1, -0.1, -0.2, -0.1, -0.2, -0.1, -0.1, -0.1, -0.2, 0.0, -0.1, -0.2, -0.1, -0.2, -0.8, -0.2, -0.1, 0.0, 0.0, -0.2, -0.1, -0.2, -0.2, -0.1, -0.2, -0.2, -0.1, -0.2, -0.1, 0.0, 0.6, 0.0, 0.0, 0.1, 0.1, 0.1, 0.0, 0.1, 0.1, 0.0, 0.1, 0.1, 0.0, 0.1, 0.0, 0.1, 0.1, 0.1, 0.0, 0.0, 0.1, 0.1, 0.1, 0.1, 0.1, 0.0, 0.0, 0.2, 0.0, 0.1, 0.2, 0.2, 0.1, 0.2, 0.1, 0.2, 0.2, 0.1, 0.2, 0.1, 0.2, 1.0, 0.0, 0.1, 0.2, 0.2, 0.1, 0.1, 0.1, 0.0, 0.1, 0.2, 0.1, -0.1, -0.2, -0.1, -0.2, -0.1, -0.2, -0.2, -0.1, -0.2, -0.1, -0.2, -0.2, -0.1, -0.2, -0.2, -0.1, -0.2, -0.1, -0.2, -0.2, -0.1, -0.2, -0.1, -0.2, -0.2, -0.1, -0.2, -0.1, -0.2, -0.2, -0.1, -0.2, -0.1, -0.2, -0.2, 0.0, 0.5, 0.0, 0.0, 0.1, 0.1, 0.0, 0.1, 0.0, 0.0, 0.0, 0.1, 0.1, 0.0, 0.1, 0.0, 0.1, 0.0, 0.0, 0.1, 0.0, 0.1, 0.0, 0.1, 0.0, 0.1, 0.0, 0.0, 0.2, 0.2, 0.0, 0.0, 0.1, 0.2, 0.0, 0.1, 0.1, 0.1, 0.1, 0.1, 0.1, 0.0, 0.2, 0.7, 0.1, 0.0, 0.1, 0.1, 0.0, 0.3, 0.1, 0.0, 0.1, -0.1, -0.1, 0.0, -0.2, -0.1, -0.1, -0.1, -0.2, 0.0, -0.1, -0.2, -0.2, 0.0, -0.1, -0.2, 0.0, -0.1, -0.2, 0.0, -0.2, -0.1, -0.2, 0.0, -0.1, -0.2, 0.0, -0.2, -0.1, -0.1, -0.1, 0.0, -0.1, -0.2, 0.0, -0.2, 0.0, 0.6, 0.0, 0.0, 0.1, 0.1, 0.0, 0.1, 0.0, 0.1, 0.1, 0.1, 0.1, 0.0, 0.1, 0.1, 0.1, 0.1, 0.1, 0.1, 0.1, 0.3, 0.1, 0.0, 0.1, 0.1, 0.0, 0.1, 0.1, -0.2, -0.2, -0.1, -0.2, -0.1, -0.2, -0.2, -0.1, -0.2, -0.1, -0.2, 0.0, 0.5, 0.0, -0.1, 0.1, 0.0, 0.0, 0.1, 0.0, 0.2, -0.2, -0.1, 0.1, 0.0, 0.2, 0.1, 0.1, 0.1, 0.1, 0.0, -0.1, -0.3, -0.2, 0.0, -0.1, 0.0, -0.2, 0.0, -0.1, 0.0, 0.0, -0.1, -0.1, 0.0, 0.0, -0.5, 0.0, 0.2, 0.1, 0.1, 0.1, 0.2, 0.0, 0.1, 0.2, 0.1, 0.1, 0.1, 0.2, 0.0, 0.1, 0.2, 0.1, 0.0, 0.2, 0.2, 0.0, 0.1, 0.2, 0.1, 0.1, 0.0, 0.0, -0.1, -0.1, -0.1, -0.1, 0.0, -0.1, 0.0, -0.1, -0.6, -0.1, 0.0, -0.2, 0.0, -0.2, 0.0, -0.1, -0.1, -0.1, 0.0, -0.1, -0.2, 0.0, -0.1, 0.0, -0.1, 0.0, -0.1, 0.0, -0.1, 0.0, 0.0, -0.1, 0.0, -0.1, 0.0, -0.1, 0.0, -0.1, 0.0, 0.0, 0.0, -0.5, 0.0, 0.1, 0.1, 0.1, 0.1, 0.1, 0.1, 0.1, 0.1, 0.2, 0.0, 0.1, 0.2, 0.1, 0.1, 0.1, 0.1, 0.1, 0.1, 0.2, 0.0, 0.2, 0.1, 0.1, 0.1, 0.1, 0.1, 0.1, 0.2, 0.1, 0.1, 0.1, 0.2, 0.0, 0.1, 0.2, 0.0, 0.1, 0.2, 0.2, 0.0, 0.1, 0.1, -0.1, 0.0, -0.1, 0.0, -0.1, -0.1, -0.3, -0.1, -0.1, 0.0, -0.1, 0.0, -0.8, -0.1, -0.1, -0.1, -0.1, -0.1, 0.0, -0.2, 0.0, -0.2, 0.0, -0.1, -0.2, 0.0, -0.1, -0.1, -0.1, 0.0, -0.2, -0.1, 0.0, -0.1, 0.0, -0.1, 0.0, -0.1, 0.0, -0.1, 0.0, -0.1, 0.0, 0.0, -0.1, -0.1, 0.0, 0.0, -0.1, 0.0, -0.1, 0.0, -0.1, 0.0, 0.0, -0.1, 0.0, -0.1, -0.1, 0.0, 0.0, -0.1, 0.0, -0.4, 0.0, 0.1, 0.1, 0.1, 0.1, 0.1, 0.2, 0.0, 0.1, 0.2, 0.0, 0.1, 0.1, 0.1, 0.0, 0.2, 0.0, 0.1, 0.2, 0.1, 0.2, 0.2, 0.0, 0.1, 0.2, 0.1, 0.0, 0.2, 0.2, 0.1, 0.2, 0.1, 0.0, 0.2, 0.1, 0.1, 0.1, 0.2, 0.2, 0.1, 0.1, 0.1, 0.1, 0.1, 0.1, 0.2, 0.1, 0.2, 0.1, 0.1, 0.1, 0.2, 0.0, 0.1, 0.2, 0.0, 0.0, -0.1, -0.1, 0.0, 0.0, -0.1, -0.1, -0.1, 0.0, 0.0, -0.1, -0.1, 0.0, -0.5, -0.1, 0.0, 0.0, -1.1, -0.1, -0.1, -0.2, -0.3, -0.1, 0.0, -0.2, 0.0, -0.2, 0.0, -0.1, -0.2, -0.1, 0.0, -0.2, -0.1, -0.1, -0.1, -0.1, -0.1, 0.0, -0.1, 0.0, -0.1, -0.1, 0.0, 0.0, -0.1, -0.1, 0.0, -0.1, 0.0, -0.1, -0.1, 0.0, 0.0, -0.1, 0.0, -0.1, -0.1, 0.0, 0.0, -0.1, -0.1, 0.0, -0.1, 0.0, -0.1, -0.1, 0.0, 0.0, -0.1, -0.1, 0.0, -0.1, 0.0, 0.0, -0.1, -0.7, -0.2, -0.1, -0.2, -0.2, -0.1, -0.2, -0.1, -0.2, -0.2, -0.1, -0.2, -0.1, -0.2, -0.2, 0.0, -0.5, 0.0, -0.1, 0.0, -0.1, -0.1, 0.0, 0.0, -0.1, 0.0, -0.1, -0.1, -0.1, -0.1, 0.0, 0.0, -0.1, 0.0, -0.1, -0.1, 0.0, 0.0, -0.1, -0.1, 0.0, -0.1, 0.0, 0.0, 0.2, 0.1, 0.2, 0.1, 0.2, 0.2, 0.1, 0.2, 0.2, 0.1, 1.8, 0.1, 0.2, 0.0, 0.2, 0.1, 0.2, 0.1, 0.2, 0.2, 0.1, 0.2, 0.1, 0.2, 0.2, 0.0, 0.0, 0.0, -0.1, -0.1, -0.1, -0.1, 0.0, -0.1, 0.0, -0.1, -0.1, -0.1, 0.0, 0.0, -0.1, -0.1, -0.1, 0.0, -0.1, 0.0, -0.1, -0.1, -0.1, -0.1, 0.0, 0.0, -0.1, -0.1, -0.2, -0.1, -0.2, -0.1, -0.2, -0.2, -0.1, -0.2, -0.1, 0.0, -0.5, -0.1, -0.1, 0.0, 0.0, -0.1, 0.0, 0.0, -0.1, -0.1, 0.0, 0.0, -0.1, -0.1, 0.0, 0.0, -0.1, 0.0, 0.0, -0.1, 0.0, -0.1, 0.2, 0.1, 0.2, 0.2, 0.1, 0.2, 0.1, 1.2, 0.1, 0.2, 0.1, 0.2, 0.0, 0.2, 0.1, 0.2, 0.1, 0.2, 0.2, 0.0, -0.1, -0.1, 0.0, -0.1, 0.0, -0.1, 0.0, 0.0, -0.1, 0.0, -0.1, 0.0, -0.1, 0.0, -0.1, 0.0, 0.0, -0.1, -0.1, 0.0, 0.0, -0.1, -0.1, 0.0, 0.0, -0.1, 0.0, -0.1, -0.1, -0.1, -0.2, -0.2, 0.0, -0.4, 0.0, -0.1, 0.0, -0.1, -0.1, -0.1, 0.0, -0.1, 0.0, -0.1, 0.0, 0.1, 0.1, 1.2, 0.1, 0.2, 0.1, 0.2, 0.0, 0.0, 0.1, -0.1, -0.1, -0.1, 0.0, -0.1, 0.0, -0.1, -0.1, 0.0, -0.1, 0.0, -0.4, 0.0, 0.0, -0.1, 0.1, 0.0, 0.2, -0.1, 0.2, 0.1, 0.0, 0.0, 0.1, 0.0, 0.1, 0.0, -0.1, 0.0, -0.1, -0.2, -0.6, -0.2, 0.1, 0.0, 0.1, 0.0, 0.1, 0.0, 0.0, 0.0, 0.5, 0.0, 0.2, 0.0, 0.1, 0.0, 0.1, 0.0, 0.1, 0.0, 0.0, 0.1, 0.0, 0.1, 0.1, 0.0, 0.0, 0.1, 0.0, 0.1, 0.0, 0.1, 0.0, 0.1, 0.0, 0.0, 0.1, 0.0, 0.0, -0.2, -0.1, -0.2, 0.0, -0.2, -0.1, -0.2, -0.1, -1.2, -0.1, -0.2, -0.1, -0.2, 0.0, 0.0, 0.0, 0.0, 0.1, 0.0, 0.1, 0.0, 0.0, 0.1, 0.0, 0.1, 0.0, 0.1, 0.0, 0.1, 0.0, 0.0, 0.1, 0.0, 0.0, 0.4, 0.0, 0.2, 0.1, 0.2, 0.2, 0.1, 0.1, 0.1, 0.0, 0.1, 0.1, 0.0, 0.1, 0.0, 0.0, 0.1, 0.1, 0.0, 0.1, 0.0, 0.0, 0.1, 0.0, 0.1, 0.0, 0.1, 0.0, 0.1, 0.0, 0.1, 0.0, 0.0, 0.1];

    PERS num y_coords_rel{5000}:=[0.0, 0.0, 0.0, 0.0, 0.0, 0.0, 0.0, 0.0, 0.0, 0.0, 0.0, 0.0, 0.0, 0.0, 0.0, 0.0, 0.0, 0.0, 0.0, 0.0, 0.0, 0.0, 0.0, 0.0, 0.0, 0.0, 0.0, 0.0, 0.0, 0.0, 0.0, 0.0, 0.0, 0.0, 0.0, 0.0, 0.0, 0.0, 0.0, 0.0, 0.0, 0.0, 0.0, 0.0, 0.0, 0.0, 0.0, 0.0, 0.0, 0.0, 0.0, 0.0, 0.0, 0.0, 0.0, 0.0, 0.0, 0.0, 0.0, 0.0, 0.0, 0.0, 0.0, 0.0, 0.0, 0.0, 0.0, 0.0, 0.0, 0.0, 0.0, 0.0, 0.0, 0.0, 0.0, 0.0, 0.0, 0.0, 0.0, 0.0, 0.0, 0.0, 0.0, 0.0, 0.0, 0.0, 0.0, 0.0, 0.0, 0.0, 0.0, 0.0, 0.0, 0.0, 0.0, 0.0, 0.0, 0.0, 0.0, 0.0, 0.0, 0.0, 0.0, 0.0, 0.0, 0.0, 0.0, 0.0, 0.0, 0.0, 0.0, 0.0, 0.0, 0.0, 0.0, 0.0, 0.0, 0.0, 0.0, 0.0, 0.0, 0.0, 0.0, 0.0, 0.0, 0.0, 0.0, 0.0, 0.0, 0.0, 0.0, 0.0, 0.0, 0.0, 0.0, 0.0, 0.0, 0.0, 0.0, 0.0, 0.0, 0.0, 0.0, 0.0, 0.0, 0.0, 0.0, 0.0, 0.0, 0.0, 0.0, 0.0, 0.0, 0.0, 0.0, 0.0, 0.0, 0.0, 0.0, 0.0, 0.0, 0.0, 0.0, 0.0, 0.0, 0.0, 0.0, 0.0, 0.0, 0.0, 0.0, 0.0, 0.0, 0.0, 0.0, 0.0, 0.0, 0.0, 0.0, 0.0, 0.0, 0.0, 0.0, 0.0, 0.0, 0.0, 0.0, 0.0, 0.0, 0.0, 0.0, 0.0, 0.0, 0.0, 0.0, 0.0, 0.0, 0.0, 0.0, 0.0, 0.0, 0.0, 0.0, 0.0, 0.0, 0.0, 0.0, 0.0, 0.0, 0.0, 0.0, 0.0, 0.0, 0.0, 0.0, 0.0, 0.0, 0.0, 0.0, 0.0, 0.0, 0.0, 0.0, 0.0, 0.0, 0.0, 0.0, 0.0, 0.0, 0.0, 0.0, 0.0, 0.0, 0.0, 0.0, 0.0, 0.0, 0.0, 0.0, 0.0, 0.0, 0.0, 0.0, 0.0, 0.0, 0.0, 0.0, 0.0, 0.0, 0.0, 0.0, 0.0, 0.0, 0.0, 0.0, 0.0, 0.0, 0.0, 0.0, 0.0, 0.0, 0.0, 0.0, 0.0, 0.0, 0.0, 0.0, 0.0, 0.0, 0.0, 0.0, 0.0, 0.0, 0.0, 0.0, 0.0, 0.0, 0.0, 0.0, 0.0, 0.0, 0.0, 0.0, 0.0, 0.0, 0.0, 0.0, 0.0, 0.0, 0.0, 0.0, 0.0, 0.0, 0.0, 0.0, 0.0, 0.0, 0.0, 0.0, 0.0, 0.0, 0.0, 0.0, 0.0, 0.0, 0.0, 0.0, 0.0, 0.0, 0.0, 0.0, 0.0, 0.0, 0.0, 0.0, 0.0, 0.0, 0.0, 0.0, 0.0, 0.0, 0.0, 0.0, 0.0, 0.0, 0.0, 0.0, 0.0, 0.0, 0.0, 0.0, 0.0, 0.0, 0.0, 0.0, 0.0, 0.0, 0.0, 0.0, 0.0, 0.0, 0.0, 0.0, 0.0, 0.0, 0.0, 0.0, 0.0, 0.0, 0.0, 0.0, 0.0, 0.0, 0.0, 0.0, 0.0, 0.0, 0.0, 0.0, 0.0, 0.0, 0.0, 0.0, 0.0, 0.0, 0.0, 0.0, 0.0, 0.0, 0.0, 0.0, 0.0, 0.0, 0.0, 0.0, 0.0, 0.0, 0.0, 0.0, 0.0, 0.0, 0.0, 0.0, 0.0, 0.0, 0.0, 0.0, 0.0, 0.0, 0.0, 0.0, 0.0, 0.0, 0.0, 0.0, 0.0, 0.0, 0.0, 0.0, 0.0, 0.0, 0.0, 0.0, 0.0, 0.0, 0.0, 0.0, 0.0, 0.0, 0.0, 0.0, 0.0, 0.0, 0.0, 0.0, 0.0, 0.0, 0.0, 0.0, 0.0, 0.0, 0.0, 0.0, 0.0, 0.0, 0.0, 0.0, 0.0, 0.0, 0.0, 0.0, 0.0, 0.0, 0.0, 0.0, 0.0, 0.0, 0.0, 0.0, 0.0, 0.0, 0.0, 0.0, 0.0, 0.0, 0.0, 0.0, 0.0, 0.0, 0.0, 0.0, 0.0, 0.0, 0.0, 0.0, 0.0, 0.0, 0.0, 0.0, 0.0, 0.0, 0.0, 0.0, 0.0, 0.0, 0.0, 0.0, 0.0, 0.0, 0.0, 0.0, 0.0, 0.0, 0.0, 0.0, 0.0, 0.0, 0.0, 0.0, 0.0, 0.0, 0.0, 0.0, 0.0, 0.0, 0.0, 0.0, 0.0, 0.0, 0.0, 0.0, 0.0, 0.0, 0.0, 0.0, 0.0, 0.0, 0.0, 0.0, 0.0, 0.0, 0.0, 0.0, 0.0, 0.0, 0.0, 0.0, 0.0, 0.0, 0.0, 0.0, 0.0, 0.0, 0.0, 0.0, 0.0, 0.0, 0.0, 0.0, 0.0, 0.0, 0.0, 0.0, 0.0, 0.0, 0.0, 0.0, 0.0, 0.0, 0.0, 0.0, 0.0, 0.0, 0.0, 0.0, 0.0, 0.0, 0.0, 0.0, 0.0, 0.0, 0.0, 0.0, 0.0, 0.0, 0.0, 0.0, 0.0, 0.0, 0.0, 0.0, 0.0, 0.0, 0.0, 0.0, 0.0, 0.0, 0.0, 0.0, 0.0, 0.0, 0.0, 0.0, 0.0, 0.0, 0.0, 0.0, 0.0, 0.0, 0.0, 0.0, 0.0, 0.0, 0.0, 0.0, 0.0, 0.0, 0.0, 0.0, 0.0, 0.0, 0.0, 0.0, 0.0, 0.0, 0.0, 0.0, 0.0, 0.0, 0.0, 0.0, 0.0, 0.0, 0.0, 0.0, 0.0, 0.0, 0.0, 0.0, 0.0, 0.0, 0.0, 0.0, 0.0, 0.0, 0.0, 0.0, 0.0, 0.0, 0.0, 0.0, 0.0, 0.0, 0.0, 0.0, 0.0, 0.0, 0.0, 0.0, 0.0, 0.0, 0.0, 0.0, 0.0, 0.0, 0.0, 0.0, 0.0, 0.0, 0.0, 0.0, 0.0, 0.0, 0.0, 0.0, 0.0, 0.0, 0.0, 0.0, 0.0, 0.0, 0.0, 0.0, 0.0, 0.0, 0.0, 0.0, 0.0, 0.0, 0.0, 0.0, 0.0, 0.0, 0.0, 0.0, 0.0, 0.0, 0.0, 0.0, 0.0, 0.0, 0.0, 0.0, 0.0, 0.0, 0.0, 0.0, 0.0, 0.0, 0.0, 0.0, 0.0, 0.0, 0.0, 0.0, 0.0, 0.0, 0.0, 0.0, 0.0, 0.0, 0.0, 0.0, 0.0, 0.0, 0.0, 0.0, 0.0, 0.0, 0.0, 0.0, 0.0, 0.0, 0.0, 0.0, 0.0, 0.0, 0.0, 0.0, 0.0, 0.0, 0.0, 0.0, 0.0, 0.0, 0.0, 0.0, 0.0, 0.0, 0.0, 0.0, 0.0, 0.0, 0.0, 0.0, 0.0, 0.0, 0.0, 0.0, 0.0, 0.0, 0.0, 0.0, 0.0, 0.0, 0.0, 0.0, 0.0, 0.0, 0.0, 0.0, 0.0, 0.0, 0.0, 0.0, 0.0, 0.0, 0.0, 0.0, 0.0, 0.0, 0.0, 0.0, 0.0, 0.0, 0.0, 0.0, 0.0, 0.0, 0.0, 0.0, 0.0, 0.0, 0.0, 0.0, 0.0, 0.0, 0.0, 0.0, 0.0, 0.0, 0.0, 0.0, 0.0, 0.0, 0.0, 0.0, 0.0, 0.0, 0.0, 0.0, 0.0, 0.0, 0.0, 0.0, 0.0, 0.0, 0.0, 0.0, 0.0, 0.0, 0.0, 0.0, 0.0, 0.0, 0.0, 0.0, 0.0, 0.0, 0.0, 0.0, 0.0, 0.0, 0.0, 0.0, 0.0, 0.0, 0.0, 0.0, 0.0, 0.0, 0.0, 0.0, 0.0, 0.0, 0.0, 0.0, 0.0, 0.0, 0.0, 0.0, 0.0, 0.0, 0.0, 0.0, 0.0, 0.0, 0.0, 0.0, 0.0, 0.0, 0.0, 0.0, 0.0, 0.0, 0.0, 0.0, 0.0, 0.0, 0.0, 0.0, 0.0, 0.0, 0.0, 0.0, 0.0, 0.0, 0.0, 0.0, 0.0, 0.0, 0.0, 0.0, 0.0, 0.0, 0.0, 0.0, 0.0, 0.0, 0.0, 0.0, 0.0, 0.0, 0.0, 0.0, 0.0, 0.0, 0.0, 0.0, 0.0, 0.0, 0.0, 0.0, 0.0, 0.0, 0.0, 0.0, 0.0, 0.0, 0.0, 0.0, 0.0, 0.0, 0.0, 0.0, 0.0, 0.0, 0.0, 0.0, 0.0, 0.0, 0.0, 0.0, 0.0, 0.0, 0.0, 0.0, 0.0, 0.0, 0.0, 0.0, 0.0, 0.0, 0.0, 0.0, 0.0, 0.0, 0.0, 0.0, 0.0, 0.0, 0.0, 0.0, 0.0, 0.0, 0.0, 0.0, 0.0, 0.0, 0.0, 0.0, 0.0, 0.0, 0.0, 0.0, 0.0, 0.0, 0.0, 0.0, 0.0, 0.0, 0.0, 0.0, 0.0, 0.0, 0.0, 0.0, 0.0, 0.0, 0.0, 0.0, 0.0, 0.0, 0.0, 0.0, 0.0, 0.0, 0.0, 0.0, 0.0, 0.0, 0.0, 0.0, 0.0, 0.0, 0.0, 0.0, 0.0, 0.0, 0.0, 0.0, 0.0, 0.0, 0.0, 0.0, 0.0, 0.0, 0.0, 0.0, 0.0, 0.0, 0.0, 0.0, 0.0, 0.0, 0.0, 0.0, 0.0, 0.0, 0.0, 0.0, 0.0, 0.0, 0.0, 0.0, 0.0, 0.0, 0.0, 0.0, 0.0, 0.0, 0.0, 0.0, 0.0, 0.0, 0.0, 0.0, 0.0, 0.0, 0.0, 0.0, 0.0, 0.0, 0.0, 0.0, 0.0, 0.0, 0.0, 0.0, 0.0, 0.0, 0.0, 0.0, 0.0, 0.0, 0.0, 0.0, 0.0, 0.0, 0.0, 0.0, 0.0, 0.0, 0.0, 0.0, 0.0, 0.0, 0.0, 0.0, 0.0, 0.0, 0.0, 0.0, 0.0, 0.0, 0.0, 0.0, 0.0, 0.0, 0.0, 0.0, 0.0, 0.0, 0.0, 0.0, 0.0, 0.0, 0.0, 0.0, 0.0, 0.0, 0.0, 0.0, 0.0, 0.0, 0.0, 0.0, 0.0, 0.0, 0.0, 0.0, 0.0, 0.0, 0.0, 0.0, 0.0, 0.0, 0.0, 0.0, 0.0, 0.0, 0.0, 0.0, 0.0, 0.0, 0.0, 0.0, 0.0, 0.0, 0.0, 0.0, 0.0, 0.0, 0.0, 0.0, 0.0, 0.0, 0.0, 0.0, 0.0, 0.0, 0.0, 0.0, 0.0, 0.0, 0.0, 0.0, 0.0, 0.0, 0.0, 0.0, 0.0, 0.0, 0.0, 0.0, 0.0, 0.0, 0.0, 0.0, 0.0, 0.0, 0.0, 0.0, 0.0, 0.0, 0.0, 0.0, 0.0, 0.0, 0.0, 0.0, 0.0, 0.0, 0.0, 0.0, 0.0, 0.0, 0.0, 0.0, 0.0, 0.0, 0.0, 0.0, 0.0, 0.0, 0.0, 0.0, 0.0, 0.0, 0.0, 0.0, 0.0, 0.0, 0.0, 0.0, 0.0, 0.0, 0.0, 0.0, 0.0, 0.0, 0.0, 0.0, 0.0, 0.0, 0.0, 0.0, 0.0, 0.0, 0.0, 0.0, 0.0, 0.0, 0.0, 0.0, 0.0, 0.0, 0.0, 0.0, 0.0, 0.0, 0.0, 0.0, 0.0, 0.0, 0.0, 0.0, 0.0, 0.0, 0.0, 0.0, 0.0, 0.0, 0.0, 0.0, 0.0, 0.0, 0.0, 0.0, 0.0, 0.0, 0.0, 0.0, 0.0, 0.0, 0.0, 0.0, 0.0, 0.0, 0.0, 0.0, 0.0, 0.0, 0.0, 0.0, 0.0, 0.0, 0.0, 0.0, 0.0, 0.0, 0.0, 0.0, 0.0, 0.0, 0.0, 0.0, 0.0, 0.0, 0.0, 0.0, 0.0, 0.0, 0.0, 0.0, 0.0, 0.0, 0.0, 0.0, 0.0, 0.0, 0.0, 0.0, 0.0, 0.0, 0.0, 0.0, 0.0, 0.0, 0.0, 0.0, 0.0, 0.0, 0.0, 0.0, 0.0, 0.0, 0.0, 0.0, 0.0, 0.0, 0.0, 0.0, 0.0, 0.0, 0.0, 0.0, 0.0, 0.0, 0.0, 0.0, 0.0, 0.0, 0.0, 0.0, 0.0, 0.0, 0.0, 0.0, 0.0, 0.0, 0.0, 0.0, 0.0, 0.0, 0.0, 0.0, 0.0, 0.0, 0.0, 0.0, 0.0, 0.0, 0.0, 0.0, 0.0, 0.0, 0.0, 0.0, 0.0, 0.0, 0.0, 0.0, 0.0, 0.0, 0.0, 0.0, 0.0, 0.0, 0.0, 0.0, 0.0, 0.0, 0.0, 0.0, 0.0, 0.0, 0.0, 0.0, 0.0, 0.0, 0.0, 0.0, 0.0, 0.0, 0.0, 0.0, 0.0, 0.0, 0.0, 0.0, 0.0, 0.0, 0.0, 0.0, 0.0, 0.0, 0.0, 0.0, 0.0, 0.0, 0.0, 0.0, 0.0, 0.0, 0.0, 0.0, 0.0, 0.0, 0.0, 0.0, 0.0, 0.0, 0.0, 0.0, 0.0, 0.0, 0.0, 0.0, 0.0, 0.0, 0.0, 0.0, 0.0, 0.0, 0.0, 0.0, 0.0, 0.0, 0.0, 0.0, 0.0, 0.0, 0.0, 0.0, 0.0, 0.0, 0.0, 0.0, 0.0, 0.0, 0.0, 0.0, 0.0, 0.0, 0.0, 0.0, 0.0, 0.0, 0.0, 0.0, 0.0, 0.0, 0.0, 0.0, 0.0, 0.0, 0.0, 0.0, 0.0, 0.0, 0.0, 0.0, 0.0, 0.0, 0.0, 0.0, 0.0, 0.0, 0.0, 0.0, 0.0, 0.0, 0.0, 0.0, 0.0, 0.0, 0.0, 0.0, 0.0, 0.0, 0.0, 0.0, 0.0, 0.0, 0.0, 0.0, 0.0, 0.0, 0.0, 0.0, 0.0, 0.0, 0.0, 0.0, 0.0, 0.0, 0.0, 0.0, 0.0, 0.0, 0.0, 0.0, 0.0, 0.0, 0.0, 0.0, 0.0, 0.0, 0.0, 0.0, 0.0, 0.0, 0.0, 0.0, 0.0, 0.0, 0.0, 0.0, 0.0, 0.0, 0.0, 0.0, 0.0, 0.0, 0.0, 0.0, 0.0, 0.0, 0.0, 0.0, 0.0, 0.0, 0.0, 0.0, 0.0, 0.0, 0.0, 0.0, 0.0, 0.0, 0.0, 0.0, 0.0, 0.0, 0.0, 0.0, 0.0, 0.0, 0.0, 0.0, 0.0, 0.0, 0.0, 0.0, 0.0, 0.0, 0.0, 0.0, 0.0, 0.0, 0.0, 0.0, 0.0, 0.0, 0.0, 0.0, 0.0, 0.0, 0.0, 0.0, 0.0, 0.0, 0.0, 0.0, 0.0, 0.0, 0.0, 0.0, 0.0, 0.0, 0.0, 0.0, 0.0, 0.0, 0.0, 0.0, 0.0, 0.0, 0.0, 0.0, 0.0, 0.0, 0.0, 0.0, 0.0, 0.0, 0.0, 0.0, 0.0, 0.0, 0.0, 0.0, 0.0, 0.0, 0.0, 0.0, 0.0, 0.0, 0.0, 0.0, 0.0, 0.0, 0.0, 0.0, 0.0, 0.0, 0.0, 0.0, 0.0, 0.0, 0.0, 0.0, 0.0, 0.0, 0.0, 0.0, 0.0, 0.0, 0.0, 0.0, 0.0, 0.0, 0.0, 0.0, 0.0, 0.0, 0.0, 0.0, 0.0, 0.0, 0.0, 0.0, 0.0, 0.0, 0.0, 0.0, 0.0, 0.0, 0.0, 0.0, 0.0, 0.0, 0.0, 0.0, 0.0, 0.0, 0.0, 0.0, 0.0, 0.0, 0.0, 0.0, 0.0, 0.0, 0.0, 0.0, 0.0, 0.0, 0.0, 0.0, 0.0, 0.0, 0.0, 0.0, 0.0, 0.0, 0.0, 0.0, 0.0, 0.0, 0.0, 0.0, 0.0, 0.0, 0.0, 0.0, 0.0, 0.0, 0.0, 0.0, 0.0, 0.0, 0.0, 0.0, 0.0, 0.0, 0.0, 0.0, 0.0, 0.0, 0.0, 0.0, 0.0, 0.0, 0.0, 0.0, 0.0, 0.0, 0.0, 0.0, 0.0, 0.0, 0.0, 0.0, 0.0, 0.0, 0.0, 0.0, 0.0, 0.0, 0.0, 0.0, 0.0, 0.0, 0.0, 0.0, 0.0, 0.0, 0.0, 0.0, 0.0, 0.0, 0.0, 0.0, 0.0, 0.0, 0.0, 0.0, 0.0, 0.0, 0.0, 0.0, 0.0, 0.0, 0.0, 0.0, 0.0, 0.0, 0.0, 0.0, 0.0, 0.0, 0.0, 0.0, 0.0, 0.0, 0.0, 0.0, 0.0, 0.0, 0.0, 0.0, 0.0, 0.0, 0.0, 0.0, 0.0, 0.0, 0.0, 0.0, 0.0, 0.0, 0.0, 0.0, 0.0, 0.0, 0.0, 0.0, 0.0, 0.0, 0.0, 0.0, 0.0, 0.0, 0.0, 0.0, 0.0, 0.0, 0.0, 0.0, 0.0, 0.0, 0.0, 0.0, 0.0, 0.0, 0.0, 0.0, 0.0, 0.0, 0.0, 0.0, 0.0, 0.0, 0.0, 0.0, 0.0, 0.0, 0.0, 0.0, 0.0, 0.0, 0.0, 0.0, 0.0, 0.0, 0.0, 0.0, 0.0, 0.0, 0.0, 0.0, 0.0, 0.0, 0.0, 0.0, 0.0, 0.0, 0.0, 0.0, 0.0, 0.0, 0.0, 0.0, 0.0, 0.0, 0.0, 0.0, 0.0, 0.0, 0.0, 0.0, 0.0, 0.0, 0.0, 0.0, 0.0, 0.0, 0.0, 0.0, 0.0, 0.0, 0.0, 0.0, 0.0, 0.0, 0.0, 0.0, 0.0, 0.0, 0.0, 0.0, 0.0, 0.0, 0.0, 0.0, 0.0, 0.0, 0.0, 0.0, 0.0, 0.0, 0.0, 0.0, 0.0, 0.0, 0.0, 0.0, 0.0, 0.0, 0.0, 0.0, 0.0, 0.0, 0.0, 0.0, 0.0, 0.0, 0.0, 0.0, 0.0, 0.0, 0.0, 0.0, 0.0, 0.0, 0.0, 0.0, 0.0, 0.0, 0.0, 0.0, 0.0, 0.0, 0.0, 0.0, 0.0, 0.0, 0.0, 0.0, 0.0, 0.0, 0.0, 0.0, 0.0, 0.0, 0.0, 0.0, 0.0, 0.0, 0.0, 0.0, 0.0, 0.0, 0.0, 0.0, 0.0, 0.0, 0.0, 0.0, 0.0, 0.0, 0.0, 0.0, 0.0, 0.0, 0.0, 0.0, 0.0, 0.0, 0.0, 0.0, 0.0, 0.0, 0.0, 0.0, 0.0, 0.0, 0.0, 0.0, 0.0, 0.0, 0.0, 0.0, 0.0, 0.0, 0.0, 0.0, 0.0, 0.0, 0.0, 0.0, 0.0, 0.0, 0.0, 0.0, 0.0, 0.0, 0.0, 0.0, 0.0, 0.0, 0.0, 0.0, 0.0, 0.0, 0.0, 0.0, 0.0, 0.0, 0.0, 0.0, 0.0, 0.0, 0.0, 0.0, 0.0, 0.0, 0.0, 0.0, 0.0, 0.0, 0.0, 0.0, 0.0, 0.0, 0.0, 0.0, 0.0, 0.0, 0.0, 0.0, 0.0, 0.0, 0.0, 0.0, 0.0, 0.0, 0.0, 0.0, 0.0, 0.0, 0.0, 0.0, 0.0, 0.0, 0.0, 0.0, 0.0, 0.0, 0.0, 0.0, 0.0, 0.0, 0.0, 0.0, 0.0, 0.0, 0.0, 0.0, 0.0, 0.0, 0.0, 0.0, 0.0, 0.0, 0.0, 0.0, 0.0, 0.0, 0.0, 0.0, 0.0, 0.0, 0.0, 0.0, 0.0, 0.0, 0.0, 0.0, 0.0, 0.0, 0.0, 0.0, 0.0, 0.0, 0.0, 0.0, 0.0, 0.0, 0.0, 0.0, 0.0, 0.0, 0.0, 0.0, 0.0, 0.0, 0.0, 0.0, 0.0, 0.0, 0.0, 0.0, 0.0, 0.0, 0.0, 0.0, 0.0, 0.0, 0.0, 0.0, 0.0, 0.0, 0.0, 0.0, 0.0, 0.0, 0.0, 0.0, 0.0, 0.0, 0.0, 0.0, 0.0, 0.0, 0.0, 0.0, 0.0, 0.0, 0.0, 0.0, 0.0, 0.0, 0.0, 0.0, 0.0, 0.0, 0.0, 0.0, 0.0, 0.0, 0.0, 0.0, 0.0, 0.0, 0.0, 0.0, 0.0, 0.0, 0.0, 0.0, 0.0, 0.0, 0.0, 0.0, 0.0, 0.0, 0.0, 0.0, 0.0, 0.0, 0.0, 0.0, 0.0, 0.0, 0.0, 0.0, 0.0, 0.0, 0.0, 0.0, 0.0, 0.0, 0.0, 0.0, 0.0, 0.0, 0.0, 0.0, 0.0, 0.0, 0.0, 0.0, 0.0, 0.0, 0.0, 0.0, 0.0, 0.0, 0.0, 0.0, 0.0, 0.0, 0.0, 0.0, 0.0, 0.0, 0.0, 0.0, 0.0, 0.0, 0.0, 0.0, 0.0, 0.0, 0.0, 0.0, 0.0, 0.0, 0.0, 0.0, 0.0, 0.0, 0.0, 0.0, 0.0, 0.0, 0.0, 0.0, 0.0, 0.0, 0.0, 0.0, 0.0, 0.0, 0.0, 0.0, 0.0, 0.0, 0.0, 0.0, 0.0, 0.0, 0.0, 0.0, 0.0, 0.0, 0.0, 0.0, 0.0, 0.0, 0.0, 0.0, 0.0, 0.0, 0.0, 0.0, 0.0, 0.0, 0.0, 0.0, 0.0, 0.0, 0.0, 0.0, 0.0, 0.0, 0.0, 0.0, 0.0, 0.0, 0.0, 0.0, 0.0, 0.0, 0.0, 0.0, 0.0, 0.0, 0.0, 0.0, 0.0, 0.0, 0.0, 0.0, 0.0, 0.0, 0.0, 0.0, 0.0, 0.0, 0.0, 0.0, 0.0, 0.0, 0.0, 0.0, 0.0, 0.0, 0.0, 0.0, 0.0, 0.0, 0.0, 0.0, 0.0, 0.0, 0.0, 0.0, 0.0, 0.0, 0.0, 0.0, 0.0, 0.0, 0.0, 0.0, 0.0, 0.0, 0.0, 0.0, 0.0, 0.0, 0.0, 0.0, 0.0, 0.0, 0.0, 0.0, 0.0, 0.0, 0.0, 0.0, 0.0, 0.0, 0.0, 0.0, 0.0, 0.0, 0.0, 0.0, 0.0, 0.0, 0.0, 0.0, 0.0, 0.0, 0.0, 0.0, 0.0, 0.0, 0.0, 0.0, 0.0, 0.0, 0.0, 0.0, 0.0, 0.0, 0.0, 0.0, 0.0, 0.0, 0.0, 0.0, 0.0, 0.0, 0.0, 0.0, 0.0, 0.0, 0.0, 0.0, 0.0, 0.0, 0.0, 0.0, 0.0, 0.0, 0.0, 0.0, 0.0, 0.0, 0.0, 0.0, 0.0, 0.0, 0.0, 0.0, 0.0, 0.0, 0.0, 0.0, 0.0, 0.0, 0.0, 0.0, 0.0, 0.0, 0.0, 0.0, 0.0, 0.0, 0.0, 0.0, 0.0, 0.0, 0.0, 0.0, 0.0, 0.0, 0.0, 0.0, 0.0, 0.0, 0.0, 0.0, 0.0, 0.0, 0.0, 0.0, 0.0, 0.0, 0.0, 0.0, 0.0, 0.0, 0.0, 0.0, 0.0, 0.0, 0.0, 0.0, 0.0, 0.0, 0.0, 0.0, 0.0, 0.0, 0.0, 0.0, 0.0, 0.0, 0.0, 0.0, 0.0, 0.0, 0.0, 0.0, 0.0, 0.0, 0.0, 0.0, 0.0, 0.0, 0.0, 0.0, 0.0, 0.0, 0.0, 0.0, 0.0, 0.0, 0.0, 0.0, 0.0, 0.0, 0.0, 0.0, 0.0, 0.0, 0.0, 0.0, 0.0, 0.0, 0.0, 0.0, 0.0, 0.0, 0.0, 0.0, 0.0, 0.0, 0.0, 0.0, 0.0, 0.0, 0.0, 0.0, 0.0, 0.0, 0.0, 0.0, 0.0, 0.0, 0.0, 0.0, 0.0, 0.0, 0.0, 0.0, 0.0, 0.0, 0.0, 0.0, 0.0, 0.0, 0.0, 0.0, 0.0, 0.0, 0.0, 0.0, 0.0, 0.0, 0.0, 0.0, 0.0, 0.0, 0.0, 0.0, 0.0, 0.0, 0.0, 0.0, 0.0, 0.0, 0.0, 0.0, 0.0, 0.0, 0.0, 0.0, 0.0, 0.0, 0.0, 0.0, 0.0, 0.0, 0.0, 0.0, 0.0, 0.0, 0.0, 0.0, 0.0, 0.0, 0.0, 0.0, 0.0, 0.0, 0.0, 0.0, 0.0, 0.0, 0.0, 0.0, 0.0, 0.0, 0.0, 0.0, 0.0, 0.0, 0.0, 0.0, 0.0, 0.0, 0.0, 0.0, 0.0, 0.0, 0.0, 0.0, 0.0, 0.0, 0.0, 0.0, 0.0, 0.0, 0.0, 0.0, 0.0, 0.0, 0.0, 0.0, 0.0, 0.0, 0.0, 0.0, 0.0, 0.0, 0.0, 0.0, 0.0, 0.0, 0.0, 0.0, 0.0, 0.0, 0.0, 0.0, 0.0, 0.0, 0.0, 0.0, 0.0, 0.0, 0.0, 0.0, 0.0, 0.0, 0.0, 0.0, 0.0, 0.0, 0.0, 0.0, 0.0, 0.0, 0.0, 0.0, 0.0, 0.0, 0.0, 0.0, 0.0, 0.0, 0.0, 0.0, 0.0, 0.0, 0.0, 0.0, 0.0, 0.0, 0.0, 0.0, 0.0, 0.0, 0.0, 0.0, 0.0, 0.0, 0.0, 0.0, 0.0, 0.0, 0.0, 0.0, 0.0, 0.0, 0.0, 0.0, 0.0, 0.0, 0.0, 0.0, 0.0, 0.0, 0.0, 0.0, 0.0, 0.0, 0.0, 0.0, 0.0, 0.0, 0.0, 0.0, 0.0, 0.0, 0.0, 0.0, 0.0, 0.0, 0.0, 0.0, 0.0, 0.0, 0.0, 0.0, 0.0, 0.0, 0.0, 0.0, 0.0, 0.0, 0.0, 0.0, 0.0, 0.0, 0.0, 0.0, 0.0, 0.0, 0.0, 0.0, 0.0, 0.0, 0.0, 0.0, 0.0, 0.0, 0.0, 0.0, 0.0, 0.0, 0.0, 0.0, 0.0, 0.0, 0.0, 0.0, 0.0, 0.0, 0.0, 0.0, 0.0, 0.0, 0.0, 0.0, 0.0, 0.0, 0.0, 0.0, 0.0, 0.0, 0.0, 0.0, 0.0, 0.0, 0.0, 0.0, 0.0, 0.0, 0.0, 0.0, 0.0, 0.0, 0.0, 0.0, 0.0, 0.0, 0.0, 0.0, 0.0, 0.0, 0.0, 0.0, 0.0, 0.0, 0.0, 0.0, 0.0, 0.0, 0.0, 0.0, 0.0, 0.0, 0.0, 0.0, 0.0, 0.0, 0.0, 0.0, 0.0, 0.0, 0.0, 0.0, 0.0, 0.0, 0.0, 0.0, 0.0, 0.0, 0.0, 0.0, 0.0, 0.0, 0.0, 0.0, 0.0, 0.0, 0.0, 0.0, 0.0, 0.0, 0.0, 0.0, 0.0, 0.0, 0.0, 0.0, 0.0, 0.0, 0.0, 0.0, 0.0, 0.0, 0.0, 0.0, 0.0, 0.0, 0.0, 0.0, 0.0, 0.0, 0.0, 0.0, 0.0, 0.0, 0.0, 0.0, 0.0, 0.0, 0.0, 0.0, 0.0, 0.0, 0.0, 0.0, 0.0, 0.0, 0.0, 0.0, 0.0, 0.0, 0.0, 0.0, 0.0, 0.0, 0.0, 0.0, 0.0, 0.0, 0.0, 0.0, 0.0, 0.0, 0.0, 0.0, 0.0, 0.0, 0.0, 0.0, 0.0, 0.0, 0.0, 0.0, 0.0, 0.0, 0.0, 0.0, 0.0, 0.0, 0.0, 0.0, 0.0, 0.0, 0.0, 0.0, 0.0, 0.0, 0.0, 0.0, 0.0, 0.0, 0.0, 0.0, 0.0, 0.0, 0.0, 0.0, 0.0, 0.0, 0.0, 0.0, 0.0, 0.0, 0.0, 0.0, 0.0, 0.0, 0.0, 0.0, 0.0, 0.0, 0.0, 0.0, 0.0, 0.0, 0.0, 0.0, 0.0, 0.0, 0.0, 0.0, 0.0, 0.0, 0.0, 0.0, 0.0, 0.0, 0.0, 0.0, 0.0, 0.0, 0.0, 0.0, 0.0, 0.0, 0.0, 0.0, 0.0, 0.0, 0.0, 0.0, 0.0, 0.0, 0.0, 0.0, 0.0, 0.0, 0.0, 0.0, 0.0, 0.0, 0.0, 0.0, 0.0, 0.0, 0.0, 0.0, 0.0, 0.0, 0.0, 0.0, 0.0, 0.0, 0.0, 0.0, 0.0, 0.0, 0.0, 0.0, 0.0, 0.0, 0.0, 0.0, 0.0, 0.0, 0.0, 0.0, 0.0, 0.0, 0.0, 0.0, 0.0, 0.0, 0.0, 0.0, 0.0, 0.0, 0.0, 0.0, 0.0, 0.0, 0.0, 0.0, 0.0, 0.0, 0.0, 0.0, 0.0, 0.0, 0.0, 0.0, 0.0, 0.0, 0.0, 0.0, 0.0, 0.0, 0.0, 0.0, 0.0, 0.0, 0.0, 0.0, 0.0, 0.0, 0.0, 0.0, 0.0, 0.0, 0.0, 0.0, 0.0, 0.0, 0.0, 0.0, 0.0, 0.0, 0.0, 0.0, 0.0, 0.0, 0.0, 0.0, 0.0, 0.0, 0.0, 0.0, 0.0, 0.0, 0.0, 0.0, 0.0, 0.0, 0.0, 0.0, 0.0, 0.0, 0.0, 0.0, 0.0, 0.0, 0.0, 0.0, 0.0, 0.0, 0.0, 0.0, 0.0, 0.0, 0.0, 0.0, 0.0, 0.0, 0.0, 0.0, 0.0, 0.0, 0.0, 0.0, 0.0, 0.0, 0.0, 0.0, 0.0, 0.0, 0.0, 0.0, 0.0, 0.0, 0.0, 0.0, 0.0, 0.0, 0.0, 0.0, 0.0, 0.0, 0.0, 0.0, 0.0, 0.0, 0.0, 0.0, 0.0, 0.0, 0.0, 0.0, 0.0, 0.0, 0.0, 0.0, 0.0, 0.0, 0.0, 0.0, 0.0, 0.0, 0.0, 0.0, 0.0, 0.0, 0.0, 0.0, 0.0, 0.0, 0.0, 0.0, 0.0, 0.0, 0.0, 0.0, 0.0, 0.0, 0.0, 0.0, 0.0, 0.0, 0.0, 0.0, 0.0, 0.0, 0.0, 0.0, 0.0, 0.0, 0.0, 0.0, 0.0, 0.0, 0.0, 0.0, 0.0, 0.0, 0.0, 0.0, 0.0, 0.0, 0.0, 0.0, 0.0, 0.0, 0.0, 0.0, 0.0, 0.0, 0.0, 0.0, 0.0, 0.0, 0.0, 0.0, 0.0, 0.0, 0.0, 0.0, 0.0, 0.0, 0.0, 0.0, 0.0, 0.0, 0.0, 0.0, 0.0, 0.0, 0.0, 0.0, 0.0, 0.0, 0.0, 0.0, 0.0, 0.0, 0.0, 0.0, 0.0, 0.0, 0.0, 0.0, 0.0, 0.0, 0.0, 0.0, 0.0, 0.0, 0.0, 0.0, 0.0, 0.0, 0.0, 0.0, 0.0, 0.0, 0.0, 0.0, 0.0, 0.0, 0.0, 0.0, 0.0, 0.0, 0.0, 0.0, 0.0, 0.0, 0.0, 0.0, 0.0, 0.0, 0.0, 0.0, 0.0, 0.0, 0.0, 0.0, 0.0, 0.0, 0.0, 0.0, 0.0, 0.0, 0.0, 0.0, 0.0, 0.0, 0.0, 0.0, 0.0, 0.0, 0.0, 0.0, 0.0, 0.0, 0.0, 0.0, 0.0, 0.0, 0.0, 0.0, 0.0, 0.0, 0.0, 0.0, 0.0, 0.0, 0.0, 0.0, 0.0, 0.0, 0.0, 0.0, 0.0, 0.0, 0.0, 0.0, 0.0, 0.0, 0.0, 0.0, 0.0, 0.0, 0.0, 0.0, 0.0, 0.0, 0.0, 0.0, 0.0, 0.0, 0.0, 0.0, 0.0, 0.0, 0.0, 0.0, 0.0, 0.0, 0.0, 0.0, 0.0, 0.0, 0.0, 0.0, 0.0, 0.0, 0.0, 0.0, 0.0, 0.0, 0.0, 0.0, 0.0, 0.0, 0.0, 0.0, 0.0, 0.0, 0.0, 0.0, 0.0, 0.0, 0.0, 0.0, 0.0, 0.0, 0.0, 0.0, 0.0, 0.0, 0.0, 0.0, 0.0, 0.0, 0.0, 0.0, 0.0, 0.0, 0.0, 0.0, 0.0, 0.0, 0.0, 0.0, 0.0, 0.0, 0.0, 0.0, 0.0, 0.0, 0.0, 0.0, 0.0, 0.0, 0.0, 0.0, 0.0, 0.0, 0.0, 0.0, 0.0, 0.0, 0.0, 0.0, 0.0, 0.0, 0.0, 0.0, 0.0, 0.0, 0.0, 0.0, 0.0, 0.0, 0.0, 0.0, 0.0, 0.0, 0.0, 0.0, 0.0, 0.0, 0.0, 0.0, 0.0, 0.0, 0.0, 0.0, 0.0, 0.0, 0.0, 0.0, 0.0, 0.0, 0.0, 0.0, 0.0, 0.0, 0.0, 0.0, 0.0, 0.0, 0.0, 0.0, 0.0, 0.0, 0.0, 0.0, 0.0, 0.0, 0.0, 0.0, 0.0, 0.0, 0.0, 0.0, 0.0, 0.0, 0.0, 0.0, 0.0, 0.0, 0.0, 0.0, 0.0, 0.0, 0.0, 0.0, 0.0, 0.0, 0.0, 0.0, 0.0, 0.0, 0.0, 0.0, 0.0, 0.0, 0.0, 0.0, 0.0, 0.0, 0.0, 0.0, 0.0, 0.0, 0.0, 0.0, 0.0, 0.0, 0.0, 0.0, 0.0, 0.0, 0.0, 0.0, 0.0, 0.0, 0.0, 0.0, 0.0, 0.0, 0.0, 0.0, 0.0, 0.0, 0.0, 0.0, 0.0, 0.0, 0.0, 0.0, 0.0, 0.0, 0.0, 0.0, 0.0, 0.0, 0.0, 0.0, 0.0, 0.0, 0.0, 0.0, 0.0, 0.0, 0.0, 0.0, 0.0, 0.0, 0.0, 0.0, 0.0, 0.0, 0.0, 0.0, 0.0, 0.0, 0.0, 0.0, 0.0, 0.0, 0.0, 0.0, 0.0, 0.0, 0.0, 0.0, 0.0, 0.0, 0.0, 0.0, 0.0, 0.0, 0.0, 0.0, 0.0, 0.0, 0.0, 0.0, 0.0, 0.0, 0.0, 0.0, 0.0, 0.0, 0.0, 0.0, 0.0, 0.0, 0.0, 0.0, 0.0, 0.0, 0.0, 0.0, 0.0, 0.0, 0.0, 0.0, 0.0, 0.0, 0.0, 0.0, 0.0, 0.0, 0.0, 0.0, 0.0, 0.0, 0.0, 0.0, 0.0, 0.0, 0.0, 0.0, 0.0, 0.0, 0.0, 0.0, 0.0, 0.0, 0.0, 0.0, 0.0, 0.0, 0.0, 0.0, 0.0, 0.0, 0.0, 0.0, 0.0, 0.0, 0.0, 0.0, 0.0, 0.0, 0.0, 0.0, 0.0, 0.0, 0.0, 0.0, 0.0, 0.0, 0.0, 0.0, 0.0, 0.0, 0.0, 0.0, 0.0, 0.0, 0.0, 0.0, 0.0, 0.0, 0.0, 0.0, 0.0, 0.0, 0.0, 0.0, 0.0, 0.0, 0.0, 0.0, 0.0, 0.0, 0.0, 0.0, 0.0, 0.0, 0.0, 0.0, 0.0, 0.0, 0.0, 0.0, 0.0, 0.0, 0.0, 0.0, 0.0, 0.0, 0.0, 0.0, 0.0, 0.0, 0.0, 0.0, 0.0, 0.0, 0.0, 0.0, 0.0, 0.0, 0.0, 0.0, 0.0, 0.0, 0.0, 0.0, 0.0, 0.0, 0.0, 0.0, 0.0, 0.0, 0.0, 0.0, 0.0, 0.0, 0.0, 0.0, 0.0, 0.0, 0.0, 0.0, 0.0, 0.0, 0.0, 0.0, 0.0, 0.0, 0.0, 0.0, 0.0, 0.0, 0.0, 0.0, 0.0, 0.0, 0.0, 0.0, 0.0, 0.0, 0.0, 0.0, 0.0, 0.0, 0.0, 0.0, 0.0, 0.0, 0.0, 0.0, 0.0, 0.0, 0.0, 0.0, 0.0, 0.0, 0.0, 0.0, 0.0, 0.0, 0.0, 0.0, 0.0, 0.0, 0.0, 0.0, 0.0, 0.0, 0.0, 0.0, 0.0, 0.0, 0.0, 0.0, 0.0, 0.0, 0.0, 0.0, 0.0, 0.0, 0.0, 0.0, 0.0, 0.0, 0.0, 0.0, 0.0, 0.0, 0.0, 0.0, 0.0, 0.0, 0.0, 0.0, 0.0, 0.0, 0.0, 0.0, 0.0, 0.0, 0.0, 0.0, 0.0, 0.0, 0.0, 0.0, 0.0, 0.0, 0.0, 0.0, 0.0, 0.0, 0.0, 0.0, 0.0, 0.0, 0.0, 0.0, 0.0, 0.0, 0.0, 0.0, 0.0, 0.0, 0.0, 0.0, 0.0, 0.0, 0.0, 0.0, 0.0, 0.0, 0.0, 0.0, 0.0, 0.0, 0.0, 0.0, 0.0, 0.0, 0.0, 0.0, 0.0, 0.0, 0.0, 0.0, 0.0, 0.0, 0.0, 0.0, 0.0, 0.0, 0.0, 0.0, 0.0, 0.0, 0.0, 0.0, 0.0, 0.0, 0.0, 0.0, 0.0, 0.0, 0.0, 0.0, 0.0, 0.0, 0.0, 0.0, 0.0, 0.0, 0.0, 0.0, 0.0, 0.0, 0.0, 0.0, 0.0, 0.0, 0.0, 0.0, 0.0, 0.0, 0.0, 0.0, 0.0, 0.0, 0.0, 0.0, 0.0, 0.0, 0.0, 0.0, 0.0, 0.0, 0.0, 0.0, 0.0, 0.0, 0.0, 0.0, 0.0, 0.0, 0.0, 0.0, 0.0, 0.0, 0.0, 0.0, 0.0, 0.0, 0.0, 0.0, 0.0, 0.0, 0.0, 0.0, 0.0, 0.0, 0.0, 0.0, 0.0, 0.0, 0.0, 0.0, 0.0, 0.0, 0.0, 0.0, 0.0, 0.0, 0.0, 0.0, 0.0, 0.0, 0.0, 0.0, 0.0, 0.0, 0.0, 0.0, 0.0, 0.0, 0.0, 0.0, 0.0, 0.0, 0.0, 0.0, 0.0, 0.0, 0.0, 0.0, 0.0, 0.0, 0.0, 0.0, 0.0, 0.0, 0.0, 0.0, 0.0, 0.0, 0.0, 0.0, 0.0, 0.0, 0.0, 0.0, 0.0, 0.0, 0.0, 0.0, 0.0, 0.0, 0.0, 0.0, 0.0, 0.0, 0.0, 0.0, 0.0, 0.0, 0.0, 0.0, 0.0, 0.0, 0.0, 0.0, 0.0, 0.0, 0.0, 0.0, 0.0, 0.0, 0.0, 0.0, 0.0, 0.0, 0.0, 0.0, 0.0, 0.0, 0.0, 0.0, 0.0, 0.0, 0.0, 0.0, 0.0, 0.0, 0.0, 0.0, 0.0, 0.0, 0.0, 0.0, 0.0, 0.0, 0.0, 0.0, 0.0, 0.0, 0.0, 0.0, 0.0, 0.0, 0.0, 0.0, 0.0, 0.0, 0.0, 0.0, 0.0, 0.0, 0.0, 0.0, 0.0, 0.0, 0.0, 0.0, 0.0, 0.0, 0.0, 0.0, 0.0, 0.0, 0.0, 0.0, 0.0, 0.0, 0.0, 0.0, 0.0, 0.0, 0.0, 0.0, 0.0, 0.0, 0.0, 0.0, 0.0, 0.0, 0.0, 0.0, 0.0, 0.0, 0.0, 0.0, 0.0, 0.0, 0.0, 0.0, 0.0, 0.0, 0.0, 0.0, 0.0, 0.0, 0.0, 0.0, 0.0, 0.0, 0.0, 0.0, 0.0, 0.0, 0.0, 0.0, 0.0, 0.0, 0.0, 0.0, 0.0, 0.0, 0.0, 0.0, 0.0, 0.0, 0.0, 0.0, 0.0, 0.0, 0.0, 0.0, 0.0, 0.0, 0.0, 0.0, 0.0, 0.0, 0.0, 0.0, 0.0, 0.0, 0.0, 0.0, 0.0, 0.0, 0.0, 0.0, 0.0, 0.0, 0.0, 0.0, 0.0, 0.0, 0.0, 0.0, 0.0, 0.0, 0.0, 0.0, 0.0, 0.0, 0.0, 0.0, 0.0, 0.0, 0.0, 0.0, 0.0, 0.0, 0.0, 0.0, 0.0, 0.0, 0.0, 0.0, 0.0, 0.0, 0.0, 0.0, 0.0, 0.0, 0.0, 0.0, 0.0, 0.0, 0.0, 0.0, 0.0, 0.0, 0.0, 0.0, 0.0, 0.0, 0.0, 0.0, 0.0, 0.0, 0.0, 0.0, 0.0, 0.0, 0.0, 0.0, 0.0, 0.0, 0.0, 0.0, 0.0, 0.0, 0.0, 0.0, 0.0, 0.0, 0.0, 0.0, 0.0, 0.0, 0.0, 0.0, 0.0, 0.0, 0.0, 0.0, 0.0, 0.0, 0.0, 0.0, 0.0, 0.0, 0.0, 0.0, 0.0, 0.0, 0.0, 0.0, 0.0, 0.0, 0.0, 0.0, 0.0, 0.0, 0.0, 0.0, 0.0, 0.0, 0.0, 0.0, 0.0, 0.0, 0.0, 0.0, 0.0, 0.0, 0.0, 0.0, 0.0, 0.0, 0.0, 0.0, 0.0, 0.0, 0.0, 0.0, 0.0, 0.0, 0.0, 0.0, 0.0, 0.0, 0.0, 0.0, 0.0, 0.0, 0.0, 0.0, 0.0, 0.0, 0.0, 0.0, 0.0, 0.0, 0.0, 0.0, 0.0, 0.0, 0.0, 0.0, 0.0, 0.0, 0.0, 0.0, 0.0, 0.0, 0.0, 0.0, 0.0, 0.0, 0.0, 0.0, 0.0, 0.0, 0.0, 0.0, 0.0, 0.0, 0.0, 0.0, 0.0, 0.0, 0.0, 0.0, 0.0, 0.0, 0.0, 0.0, 0.0, 0.0, 0.0, 0.0, 0.0, 0.0, 0.0, 0.0, 0.0, 0.0, 0.0, 0.0, 0.0, 0.0, 0.0, 0.0, 0.0, 0.0, 0.0, 0.0, 0.0, 0.0, 0.0, 0.0, 0.0, 0.0, 0.0, 0.0, 0.0, 0.0, 0.0, 0.0, 0.0, 0.0, 0.0, 0.0, 0.0, 0.0, 0.0, 0.0, 0.0, 0.0, 0.0, 0.0, 0.0, 0.0, 0.0, 0.0, 0.0, 0.0, 0.0, 0.0, 0.0, 0.0, 0.0, 0.0, 0.0, 0.0, 0.0, 0.0, 0.0, 0.0, 0.0, 0.0, 0.0, 0.0, 0.0, 0.0, 0.0, 0.0, 0.0, 0.0, 0.0, 0.0, 0.0, 0.0, 0.0, 0.0, 0.0, 0.0, 0.0, 0.0, 0.0, 0.0, 0.0, 0.0, 0.0, 0.0, 0.0, 0.0, 0.0, 0.0, 0.0, 0.0, 0.0, 0.0, 0.0, 0.0, 0.0, 0.0, 0.0, 0.0, 0.0, 0.0, 0.0, 0.0, 0.0, 0.0, 0.0, 0.0, 0.0, 0.0, 0.0, 0.0, 0.0, 0.0, 0.0, 0.0, 0.0, 0.0, 0.0, 0.0, 0.0, 0.0, 0.0, 0.0, 0.0, 0.0, 0.0, 0.0, 0.0, 0.0, 0.0, 0.0, 0.0, 0.0, 0.0, 0.0, 0.0, 0.0, 0.0, 0.0, 0.0, 0.0, 0.0, 0.0, 0.0, 0.0, 0.0, 0.0, 0.0, 0.0, 0.0, 0.0, 0.0, 0.0, 0.0, 0.0, 0.0, 0.0, 0.0, 0.0, 0.0, 0.0, 0.0, 0.0, 0.0, 0.0, 0.0, 0.0, 0.0, 0.0, 0.0, 0.0, 0.0, 0.0, 0.0, 0.0, 0.0, 0.0, 0.0, 0.0, 0.0, 0.0, 0.0, 0.0, 0.0, 0.0, 0.0, 0.0, 0.0, 0.0, 0.0, 0.0, 0.0, 0.0, 0.0, 0.0, 0.0, 0.0, 0.0, 0.0, 0.0, 0.0, 0.0, 0.0, 0.0, 0.0, 0.0, 0.0, 0.0, 0.0, 0.0, 0.0, 0.0, 0.0, 0.0, 0.0, 0.0, 0.0, 0.0, 0.0, 0.0, 0.0, 0.0, 0.0, 0.0, 0.0, 0.0, 0.0, 0.0, 0.0, 0.0, 0.0, 0.0, 0.0, 0.0, 0.0, 0.0, 0.0, 0.0, 0.0, 0.0, 0.0, 0.0, 0.0, 0.0, 0.0, 0.0, 0.0, 0.0, 0.0, 0.0, 0.0, 0.0, 0.0, 0.0, 0.0, 0.0, 0.0, 0.0, 0.0, 0.0, 0.0, 0.0, 0.0, 0.0, 0.0, 0.0, 0.0, 0.0, 0.0, 0.0, 0.0, 0.0, 0.0, 0.0, 0.0, 0.0, 0.0, 0.0, 0.0, 0.0, 0.0, 0.0, 0.0, 0.0, 0.0, 0.0, 0.0, 0.0, 0.0, 0.0, 0.0, 0.0, 0.0, 0.0, 0.0, 0.0, 0.0, 0.0, 0.0, 0.0, 0.0, 0.0, 0.0, 0.0, 0.0, 0.0, 0.0, 0.0, 0.0, 0.0, 0.0, 0.0, 0.0, 0.0, 0.0, 0.0, 0.0, 0.0, 0.0, 0.0, 0.0, 0.0, 0.0, 0.0, 0.0, 0.0, 0.0, 0.0, 0.0, 0.0, 0.0, 0.0, 0.0, 0.0, 0.0, 0.0, 0.0, 0.0, 0.0, 0.0, 0.0, 0.0, 0.0, 0.0, 0.0, 0.0, 0.0, 0.0, 0.0, 0.0, 0.0, 0.0, 0.0, 0.0, 0.0, 0.0, 0.0, 0.0, 0.0, 0.0, 0.0, 0.0, 0.0, 0.0, 0.0, 0.0, 0.0, 0.0, 0.0, 0.0, 0.0, 0.0, 0.0, 0.0, 0.0, 0.0, 0.0, 0.0, 0.0, 0.0, 0.0, 0.0, 0.0, 0.0, 0.0, 0.0, 0.0, 0.0, 0.0, 0.0, 0.0, 0.0, 0.0, 0.0, 0.0, 0.0, 0.0, 0.0, 0.0, 0.0, 0.0, 0.0, 0.0, 0.0, 0.0, 0.0, 0.0, 0.0, 0.0, 0.0, 0.0, 0.0, 0.0, 0.0, 0.0, 0.0, 0.0, 0.0, 0.0, 0.0, 0.0, 0.0, 0.0, 0.0, 0.0, 0.0, 0.0, 0.0, 0.0, 0.0, 0.0, 0.0, 0.0, 0.0, 0.0, 0.0, 0.0, 0.0, 0.0, 0.0, 0.0, 0.0, 0.0, 0.0, 0.0, 0.0, 0.0, 0.0, 0.0, 0.0, 0.0, 0.0, 0.0, 0.0, 0.0, 0.0, 0.0, 0.0, 0.0, 0.0, 0.0, 0.0, 0.0, 0.0, 0.0, 0.0, 0.0, 0.0, 0.0, 0.0, 0.0, 0.0, 0.0, 0.0, 0.0, 0.0, 0.0, 0.0, 0.0, 0.0, 0.0, 0.0, 0.0, 0.0, 0.0, 0.0, 0.0, 0.0, 0.0, 0.0, 0.0, 0.0, 0.0, 0.0, 0.0, 0.0, 0.0, 0.0, 0.0, 0.0, 0.0, 0.0, 0.0, 0.0, 0.0, 0.0, 0.0, 0.0, 0.0, 0.0, 0.0, 0.0, 0.0, 0.0, 0.0, 0.0, 0.0, 0.0, 0.0, 0.0, 0.0, 0.0, 0.0, 0.0, 0.0, 0.0, 0.0, 0.0, 0.0, 0.0, 0.0, 0.0, 0.0, 0.0, 0.0, 0.0, 0.0, 0.0, 0.0, 0.0, 0.0, 0.0, 0.0, 0.0, 0.0, 0.0, 0.0, 0.0, 0.0, 0.0, 0.0, 0.0, 0.0, 0.0, 0.0, 0.0, 0.0, 0.0, 0.0, 0.0, 0.0, 0.0, 0.0, 0.0, 0.0, 0.0, 0.0, 0.0, 0.0, 0.0, 0.0, 0.0, 0.0, 0.0, 0.0, 0.0, 0.0, 0.0, 0.0, 0.0, 0.0, 0.0, 0.0, 0.0, 0.0, 0.0, 0.0, 0.0, 0.0, 0.0, 0.0, 0.0, 0.0, 0.0, 0.0, 0.0, 0.0, 0.0, 0.0, 0.0, 0.0, 0.0, 0.0, 0.0, 0.0, 0.0, 0.0, 0.0, 0.0, 0.0, 0.0, 0.0, 0.0, 0.0, 0.0, 0.0, 0.0, 0.0, 0.0, 0.0, 0.0, 0.0, 0.0, 0.0, 0.0, 0.0, 0.0, 0.0, 0.0, 0.0, 0.0, 0.0, 0.0, 0.0, 0.0, 0.0, 0.0, 0.0, 0.0, 0.0, 0.0, 0.0, 0.0, 0.0, 0.0, 0.0, 0.0, 0.0, 0.0, 0.0, 0.0, 0.0, 0.0, 0.0, 0.0, 0.0, 0.0, 0.0, 0.0, 0.0, 0.0, 0.0, 0.0, 0.0, 0.0, 0.0, 0.0, 0.0, 0.0, 0.0, 0.0, 0.0, 0.0, 0.0, 0.0, 0.0, 0.0, 0.0, 0.0, 0.0, 0.0, 0.0, 0.0, 0.0, 0.0, 0.0, 0.0, 0.0, 0.0, 0.0, 0.0, 0.0, 0.0, 0.0, 0.0, 0.0, 0.0, 0.0, 0.0, 0.0, 0.0, 0.0, 0.0, 0.0, 0.0, 0.0, 0.0, 0.0, 0.0, 0.0, 0.0, 0.0, 0.0, 0.0, 0.0, 0.0, 0.0, 0.0, 0.0, 0.0, 0.0, 0.0, 0.0, 0.0, 0.0, 0.0, 0.0, 0.0, 0.0, 0.0, 0.0, 0.0, 0.0, 0.0, 0.0, 0.0, 0.0, 0.0, 0.0, 0.0, 0.0, 0.0, 0.0, 0.0, 0.0, 0.0, 0.0, 0.0, 0.0, 0.0, 0.0, 0.0, 0.0, 0.0, 0.0, 0.0, 0.0, 0.0, 0.0, 0.0, 0.0, 0.0, 0.0, 0.0, 0.0, 0.0, 0.0, 0.0, 0.0, 0.0, 0.0, 0.0, 0.0, 0.0, 0.0, 0.0, 0.0, 0.0, 0.0, 0.0, 0.0, 0.0, 0.0, 0.0, 0.0, 0.0, 0.0, 0.0, 0.0, 0.0, 0.0, 0.0, 0.0, 0.0, 0.0, 0.0, 0.0, 0.0, 0.0, 0.0, 0.0, 0.0, 0.0, 0.0, 0.0, 0.0, 0.0, 0.0, 0.0, 0.0, 0.0, 0.0, 0.0, 0.0, 0.0, 0.0, 0.0, 0.0, 0.0, 0.0, 0.0, 0.0, 0.0, 0.0, 0.0, 0.0, 0.0, 0.0, 0.0, 0.0, 0.0, 0.0, 0.0, 0.0, 0.0, 0.0, 0.0, 0.0, 0.0, 0.0, 0.0, 0.0, 0.0, 0.0, 0.0, 0.0, 0.0, 0.0, 0.0, 0.0, 0.0, 0.0, 0.0, 0.0, 0.0, 0.0, 0.0, 0.0, 0.0, 0.0, 0.0, 0.0, 0.0, 0.0, 0.0, 0.0, 0.0, 0.0, 0.0, 0.0, 0.0, 0.0, 0.0, 0.0, 0.0, 0.0, 0.0, 0.0, 0.0, 0.0, 0.0, 0.0, 0.0, 0.0, 0.0, 0.0, 0.0, 0.0, 0.0, 0.0, 0.0, 0.0, 0.0, 0.0, 0.0, 0.0, 0.0, 0.0, 0.0, 0.0, 0.0, 0.0, 0.0, 0.0, 0.0, 0.0, 0.0, 0.0, 0.0, 0.0, 0.0, 0.0, 0.0, 0.0, 0.0, 0.0, 0.0, 0.0, 0.0, 0.0, 0.0, 0.0];

    PERS num z_coords_rel{5000}:=[0.0, -0.1, -0.2, -0.1, -0.2, -0.2, -0.1, -0.2, -0.2, -0.1, -0.2, -0.1, -0.2, -0.2, -0.1, -0.2, -0.1, -0.2, -0.2, -0.1, -0.2, -0.1, -0.2, -0.2, -0.1, -0.2, -0.1, -0.2, -0.2, -0.1, -0.2, -0.1, 0.0, -0.2, 0.0, 0.0, -0.2, -0.1, -0.2, -0.2, -0.1, -0.2, -0.1, -0.2, -0.2, -0.1, -0.2, -0.1, -0.2, -0.2, -0.1, -0.2, -0.1, -0.2, -0.2, -0.1, -0.2, -0.1, -0.2, -0.2, -0.1, -0.2, -0.1, -0.2, -0.2, -0.1, -0.2, -0.2, -0.1, -0.2, -0.1, -0.2, -0.2, 0.0, -0.1, 0.0, 0.0, -0.2, -0.1, -0.2, -0.2, -0.1, -0.2, -0.1, -0.2, -0.2, -0.1, -0.2, -0.1, -0.2, -0.2, -0.1, -0.2, -0.2, -0.1, -0.2, -0.1, -0.2, -0.2, -0.1, -0.2, -0.1, -0.2, -0.2, -0.1, -0.2, -0.1, -0.2, -0.2, -0.1, -0.2, -0.1, -0.2, -0.2, -0.1, 0.0, -0.2, 0.0, 0.0, -0.1, -0.2, -0.2, -0.1, -0.2, -0.2, -0.1, -0.2, -0.1, -0.2, -0.2, -0.1, -0.2, -0.1, -0.2, -0.2, -0.1, -0.2, -0.1, -0.2, -0.2, -0.1, -0.2, -0.1, -0.2, -0.2, -0.1, -0.2, -0.2, -0.1, -0.2, -0.1, -0.2, -0.2, -0.1, -0.2, -0.1, -0.2, -0.2, 0.0, -0.1, 0.0, 0.0, -0.2, -0.1, -0.2, -0.2, -0.1, -0.2, -0.1, -0.2, -0.2, -0.1, -0.2, -0.1, -0.2, -0.2, -0.1, -0.2, -0.2, -0.1, -0.2, -0.1, -0.2, -0.2, -0.1, -0.2, -0.1, -0.2, -0.2, -0.1, -0.2, -0.1, -0.2, -0.2, -0.1, -0.2, -0.1, -0.2, -0.2, -0.1, -0.2, -0.2, 0.0, 0.0, 0.0, 0.2, 0.0, 0.2, 0.0, 0.1, 0.0, 0.2, 0.0, -0.2, 0.0, 0.0, -0.1, 0.0, -0.2, 0.0, -0.2, 0.0, -0.1, 0.0, 0.0, -0.2, -0.1, -0.2, -0.2, -0.1, -0.2, -0.1, -0.2, -0.2, -0.1, -0.2, -0.1, -0.2, -0.2, -0.1, -0.2, -0.1, -0.2, -0.2, 0.0, -0.9, 0.0, -1.0, 0.0, -1.1, 0.0, -0.2, 0.0, 1.1, 0.0, 1.0, 0.0, 1.0, 0.0, 0.1, 0.2, 0.2, 0.0, 0.0, -0.2, 0.0, -0.2, 0.0, -0.1, -0.2, 0.0, -0.1, 0.0, -0.2, -0.2, -2.1, -0.1, -2.1, -0.2, -0.9, -0.2, 0.0, -0.2, 0.0, 0.0, -0.1, 0.0, 0.0, -0.2, 0.0, -0.1, -0.2, 0.2, 0.0, 0.1, 0.0, 0.0, 0.2, 0.0, 0.0, 0.1, 0.0, 0.0, -0.1, 0.0, -0.2, 0.0, 0.0, -0.1, 0.0, -0.2, 0.0, -0.2, 0.0, 0.0, -0.1, 0.0, -0.2, 0.0, -0.1, -0.2, -0.2, -0.1, -1.8, -0.2, -1.6, -0.1, -0.8, -0.2, -0.1, 0.0, -0.2, 0.0, -0.2, 0.0, -0.1, 0.0, -0.2, 0.0, -0.2, 0.0, -0.1, 0.1, 0.2, 0.0, 0.2, 0.1, 0.2, 0.0, 0.6, 0.0, 0.7, 0.0, 0.1, 0.2, 0.2, 0.0, 0.8, 0.1, 0.2, 0.1, 0.2, 0.2, 0.1, 0.2, 0.1, 0.2, 0.2, 0.1, 0.2, 0.2, 0.1, 0.2, 0.1, 0.0, -0.1, -0.2, -0.1, -0.2, -0.2, -0.1, -0.2, -0.2, -0.1, -0.2, -0.1, -0.2, -0.2, -0.1, -0.2, -0.1, -0.2, 0.0, -0.2, 0.0, 0.0, -0.1, 0.0, -0.2, 0.0, -0.1, 0.0, -0.2, 0.0, 0.0, -0.2, 0.0, -0.1, 0.0, -0.2, 0.0, 3.2, 0.0, -3.3, -0.2, -0.2, -0.1, -0.2, -0.1, -0.2, -0.2, -0.1, -0.2, -0.2, -0.1, -0.2, -0.1, -0.2, -0.2, -0.1, 0.0, -0.2, 0.0, -0.1, -0.2, 0.0, -0.2, 0.0, -0.1, 0.0, -0.2, 0.0, -0.1, 0.0, -0.2, 0.0, -0.2, 0.0, -0.1, 0.0, 0.0, 0.1, 0.0, 0.2, 0.0, 0.2, 0.0, 0.1, 0.0, 0.2, 0.0, 0.1, 0.0, 0.2, 0.0, 0.2, 0.1, 0.0, 0.2, 0.0, 0.1, 0.0, 0.2, 0.0, 0.0, -0.2, 0.0, -0.1, 0.0, -0.2, 0.0, -0.1, 0.0, -0.2, -0.2, 0.0, -0.1, 0.0, -0.2, 0.0, -0.1, 0.0, -0.2, 0.0, -0.2, 0.0, -0.1, 0.0, -0.2, -4.6, -0.9, 0.0, -0.1, 0.0, 0.0, -0.2, -0.1, -0.2, -0.2, -0.8, -0.1, -0.7, -0.1, -0.8, -0.2, -0.79, -0.16, -0.65, -0.16, -0.16, -0.16, -0.16, -0.16, -0.16, 0.0, -0.16, -0.16, -0.16, 0.0, -0.16, -0.17, -0.16, 0.0, -0.16, -0.16, -0.16, 0.0, -0.16, 0.0, 0.16, 0.16, 0.16, 0.0, 0.16, 0.16, 0.17, 0.0, 0.16, 0.16, 0.16, 0.0, 0.16, 0.16, 0.16, 1.29, 0.16, 0.79, 0.2, 0.8, 0.1, 0.7, 0.1, 0.8, 0.2, 0.6, 0.7, 0.0, 4.7, 0.1, 0.2, 0.0, 0.1, 0.0, 0.2, 0.0, 0.2, 0.0, 0.1, 0.0, 0.2, 0.0, 0.1, 0.0, 0.2, 0.2, 0.0, 0.1, 0.0, 0.2, 0.6, 0.2, 0.1, 0.2, 0.2, 0.1, 0.2, 0.2, 0.1, 0.2, 0.1, 0.2, 0.2, 0.1, 0.0, 0.2, 0.0, 0.1, 0.0, 0.0, 0.2, 0.0, 0.2, 0.0, 0.1, 0.0, 0.2, 0.0, 0.0, 0.1, 0.0, 0.2, 0.0, -0.2, 0.0, -0.6, 0.0, -0.2, -0.1, -0.2, 0.0, -0.6, 0.0, -0.7, 0.0, -0.1, -0.2, -0.2, 0.0, -0.1, -0.2, -0.1, -0.2, -0.2, -0.1, -0.2, -0.1, -0.2, -0.2, -0.1, -0.2, -0.1, -0.2, -0.2, -0.1, -0.2, -0.1, -0.2, -0.2, -0.1, 0.0, -0.2, 0.0, 0.0, 0.0, -0.2, 0.0, 0.0, -0.1, 0.0, 0.0, -0.2, 0.0, 0.0, -0.1, 0.0, 0.0, -0.2, 0.0, 0.0, 0.2, 0.0, 0.0, 0.1, 0.0, 0.0, 0.2, 0.0, 0.0, 0.1, 0.0, 0.0, 0.0, 0.2, 0.0, 0.0, 0.8, 0.2, 0.1, 0.2, 0.2, 0.1, 0.2, 0.1, 0.2, 0.2, 0.1, 0.2, 0.1, 0.2, 0.2, 0.1, 0.2, 0.0, 0.1, 0.0, 0.2, 0.0, 0.2, 0.0, 0.1, 0.0, 0.2, 0.0, 0.2, 0.0, 0.0, -0.2, 0.0, -0.2, 0.0, 0.0, -0.1, 0.0, -0.2, 0.0, 0.0, -0.2, 0.0, -0.1, 0.0, 0.0, -0.2, 0.0, -0.1, -0.2, -0.2, -0.1, -0.2, -0.1, -0.2, -0.2, -0.1, -0.2, -0.1, -0.2, -0.2, -0.1, -0.2, -0.1, -0.2, -0.2, -0.1, -0.2, -0.2, -0.1, -0.2, -0.1, -0.2, -0.2, -0.1, -0.2, -0.1, -0.2, -0.2, -0.1, 0.0, 0.0, -0.2, 0.0, 0.0, -0.1, 0.0, 0.0, 0.0, -0.2, 0.0, 0.0, 0.0, -0.2, 0.0, 0.0, -0.1, 0.0, 0.0, 0.0, -0.2, 0.0, 0.0, -0.1, 0.0, 0.0, 0.1, 0.0, 0.0, 0.0, 0.2, 0.0, 0.0, 0.1, 0.0, 0.0, 0.0, 0.2, 0.0, 0.0, 0.0, 0.2, 0.0, 0.0, 0.1, 0.0, 0.0, 0.0, -0.1, -0.2, -0.2, -0.1, -0.2, -0.1, -0.2, -0.2, -0.1, -0.2, -0.1, -0.2, -0.2, -0.1, -0.2, -0.2, -0.1, -0.2, -0.1, -0.2, -0.2, -0.1, -0.2, -0.1, -0.2, -0.2, -0.1, -0.2, -0.1, -0.2, -0.2, -0.1, -0.2, -0.1, -0.2, -0.2, -0.1, -0.2, -0.1, -0.2, -0.2, -0.13, -0.16, -0.16, -0.16, -0.17, -0.16, -0.16, -0.16, 0.0, -0.16, 0.0, 0.0, -0.16, 0.0, 0.0, 0.16, 0.0, 0.64, 0.17, 0.16, 0.16, 0.16, 0.13, 0.2, 0.2, 0.1, 0.2, 0.1, 0.2, 0.2, 0.1, 0.2, 0.1, 0.2, 0.2, 0.1, 0.2, 0.1, 0.7, 0.1, 0.2, 0.2, 0.1, 0.2, 0.1, 0.2, 0.2, 0.1, 0.2, 0.2, 0.1, 0.2, 0.1, 0.2, 0.2, 0.1, 0.2, 0.1, 0.2, 0.2, 0.1, 0.2, 0.1, 0.2, 0.2, 0.1, 0.0, 0.0, 0.0, 0.2, 0.0, 0.1, 0.0, 0.0, 0.0, 0.2, 0.0, 0.0, 0.0, 0.2, 0.0, 0.1, 0.0, 0.0, 0.0, 0.2, 0.0, 0.0, 0.0, 0.1, 0.0, 0.2, 0.0, -0.2, 0.0, 0.0, 0.0, -0.1, 0.0, 0.0, 0.0, -0.2, 0.0, -0.1, 0.0, 0.0, 0.0, -0.2, 0.0, 0.0, 0.0, -0.2, 0.0, -0.1, 0.0, 0.0, 0.0, 0.1, 0.2, 0.2, 0.1, 0.2, 0.1, 0.2, 0.2, 0.1, 0.2, 0.2, 0.1, 0.2, 0.1, 0.2, 0.2, 0.1, 0.2, 0.1, 0.2, 0.2, 0.1, 0.2, 0.1, 0.2, 0.2, 0.8, 0.0, 1.1, 0.0, 1.0, 0.0, 0.1, 0.0, -0.9, 0.0, -1.2, 0.0, -0.8, 0.0, 0.0, 0.2, 0.0, 0.1, 0.0, 0.0, 0.2, 0.0, 0.2, 0.0, 0.0, 0.1, 0.0, 0.2, 0.0, 0.0, 0.2, 0.0, 0.1, 0.0, 0.2, 0.8, 0.1, 1.6, 0.2, 1.8, 0.1, 0.2, 0.2, 0.1, 0.0, 0.2, 0.0, 0.1, 0.0, 0.2, 0.0, -0.2, 0.0, -0.1, 0.0, -0.2, 0.0, 0.0, 0.2, 0.0, 0.1, 0.0, 0.2, 0.0, 0.0, 0.2, 0.0, 0.1, 0.0, 0.2, 0.0, 0.0, 0.1, 0.0, 0.2, 0.0, 0.2, 0.9, 0.2, 2.1, 0.1, 2.0, 0.1, 0.0, 0.0, 0.2, 0.0, 0.2, 0.0, 0.1, 0.0, 0.2, 0.1, -0.1, 0.0, -0.2, 0.0, -0.1, 0.0, -0.2, 0.0, 0.2, 0.1, 0.0, 0.2, 0.0, 0.1, 0.2, 0.0, 0.2, 0.0, 0.1, 0.2, 0.1, 0.2, 0.2, 0.1, 0.2, 0.1, 0.2, 0.2, 0.1, 0.2, 0.1, 0.2, 0.2, 0.1, 0.2, 0.1, 0.2, 0.2, 0.1, 0.2, 0.2, 0.1, 0.2, 0.1, 0.2, 0.2, 0.1, 0.2, 0.1, 0.2, 0.2, 0.1, 0.2, 0.1, 0.2, 0.0, 0.2, 0.0, 0.1, 0.2, 0.1, 0.2, 0.2, 0.1, 0.2, 0.2, 0.1, 0.2, 0.1, 0.2, 0.2, 0.1, 0.2, 0.1, 0.2, 0.2, 0.1, 0.2, 0.1, 0.2, 0.2, 0.1, 0.2, 0.1, 0.2, 0.2, 0.1, 0.2, 0.1, 0.2, 0.2, 0.1, 0.2, 0.2, 0.1, 0.2, 0.1, 0.2, 0.0, 0.2, 0.0, 0.1, 0.2, 0.1, 0.2, 0.2, 0.1, 0.2, 0.1, 0.2, 0.2, 0.1, 0.2, 0.1, 0.2, 0.2, 0.1, 0.2, 0.2, 0.1, 0.2, 0.1, 0.2, 0.2, 0.1, 0.2, 0.1, 0.2, 0.2, 0.1, 0.2, 0.1, 0.2, 0.2, 0.1, 0.2, 0.1, 0.2, 0.2, 0.1, 0.2, 0.0, 0.1, 0.0, 0.2, 0.2, 0.1, 0.2, 0.2, 0.1, 0.2, 0.1, 0.2, 0.2, 0.1, 0.2, 0.1, 0.2, 0.2, 0.1, 0.2, 0.1, 0.2, 0.2, 0.1, 0.2, 0.1, 0.2, 0.2, 0.1, 0.2, 0.2, 0.1, 0.2, 0.1, 0.2, 0.2, 0.1, 0.2, 0.1, 0.2, 0.2, 0.0, 0.1, 0.0, 0.2, 0.1, 0.2, 0.2, 0.1, 0.2, 0.1, 0.2, 0.2, 0.1, 0.2, 0.1, 0.2, 0.2, 0.1, 0.2, 0.2, 0.1, 0.2, 0.1, 0.2, 0.2, 0.1, 0.2, 0.1, 0.2, 0.2, 0.1, 0.2, 0.1, 0.2, 0.2, 0.1, 0.2, 0.1, 0.2, 0.2, 0.1, 0.0, 0.2, 0.0, 0.1, 0.2, 0.2, 0.1, 0.2, 0.2, 0.1, 0.2, 0.1, 0.2, 0.2, 0.1, 0.2, 0.1, 0.2, 0.2, 0.1, 0.2, 0.1, 0.2, 0.2, 0.1, 0.2, 0.1, 0.2, 0.2, 0.1, 0.2, 0.2, 0.1, 0.2, 0.1, 0.0, -0.1, -0.2, -0.1, -0.2, -0.2, -0.1, -0.2, -0.2, -0.1, -0.2, -0.1, -0.2, -0.2, -0.1, -0.2, -0.1, -0.2, 0.0, 0.2, 4.8, 0.1, 0.0, 0.2, 0.0, 0.2, 0.0, 0.1, 0.2, -0.2, 0.0, -0.1, 0.0, -0.2, 0.0, 0.2, 5.0, 0.1, 0.0, 0.0, 0.2, 0.0, 0.0, 0.1, 0.0, 0.0, 0.2, 0.0, 0.2, 0.0, 0.0, 0.1, 0.0, 0.2, 0.0, -0.2, 0.0, 0.0, -0.1, 0.0, -0.2, 0.0, 0.0, -0.2, 0.0, 0.0, -0.1, 0.0, 0.0, -0.2, 0.2, 0.1, 0.0, 0.7, 0.1, 0.7, 0.1, 0.2, 0.2, 0.1, 0.2, 0.1, 0.2, 0.2, 0.1, 0.2, 0.1, 0.2, 0.2, 0.1, 0.2, 0.2, 0.1, 0.2, 0.1, 0.2, 0.2, 0.1, 0.2, 0.0, 0.0, 0.0, 0.1, 0.0, 0.0, 0.0, 0.2, 0.0, 0.0, 0.2, 0.0, 0.0, 0.0, 0.1, 0.0, 0.0, 0.0, 0.2, 0.0, 0.0, 0.1, 0.0, 0.0, 0.0, 0.2, 0.0, 0.0, 0.0, 0.2, 0.0, 0.0, 0.1, 0.0, 0.0, -0.1, 0.0, 0.0, 0.0, -0.2, 0.0, 0.0, 0.0, -0.2, 0.0, 0.0, -0.1, 0.0, 0.0, 0.0, -0.2, 0.0, 0.0, 0.0, -0.1, 0.0, 0.0, -0.2, 0.0, 0.0, 0.0, -0.2, 0.0, 0.0, 0.0, -0.1, 0.0, 0.1, 0.7, 0.1, 3.3, 0.1, 0.7, 0.1, 0.2, 0.1, 0.2, 0.2, 0.1, 0.2, 0.1, 0.2, 0.2, 0.1, 0.2, 0.2, 0.1, 0.2, 0.0, 0.0, 0.8, 0.1, 0.2, 0.2, 0.1, 0.7, 0.1, 1.0, 0.0, 0.6, 0.0, 0.2, 0.2, 0.0, 0.1, 0.0, 0.2, 0.0, 0.1, 0.0, 0.2, 0.0, 0.2, 0.0, 0.1, 0.0, -0.1, -0.2, -0.2, -0.1, -0.2, -0.1, -0.2, -0.2, -0.1, -0.2, -0.2, -0.1, -0.2, -0.1, -0.2, -0.2, -0.1, -0.2, -0.1, -0.2, -0.2, -0.1, -0.2, -0.1, -0.2, -0.2, -0.1, -0.2, -0.1, -0.2, -0.2, -0.1, -0.2, 0.0, 0.2, 0.1, 0.2, 0.2, 0.1, 0.2, 0.1, 0.2, 0.2, 0.1, 0.2, 0.1, 0.2, 0.2, 0.1, 0.2, 0.1, 0.2, 0.2, 0.1, 0.2, 0.1, 0.2, 0.2, 0.1, 0.2, 0.2, 0.1, 0.2, 0.1, 0.2, 0.2, 0.1, 0.2, 0.0, 0.0, 0.0, 0.1, 0.0, 0.0, 0.0, 0.2, 0.0, 0.0, 0.0, 0.0, 0.0, 0.0, -0.2, 0.0, -0.1, 0.0, 0.0, -0.2, 0.0, 0.0, -0.1, -0.2, -0.2, -0.1, -0.2, -0.1, -0.2, -0.2, -0.1, -0.2, -0.2, -0.1, -0.2, -0.1, -0.2, -0.2, -0.1, -0.2, -0.1, -0.2, -0.2, -0.1, -0.2, -0.1, -0.2, -0.2, -0.1, -0.2, -0.1, -0.2, -0.2, -0.1, -0.2, -0.1, 0.0, 0.1, 0.2, 0.1, 0.2, 0.2, 0.1, 0.2, 0.1, 0.2, 0.2, 0.1, 0.2, 0.1, 0.2, 0.2, 0.1, 0.2, 0.1, 0.2, 0.2, 0.1, 0.2, 0.1, 0.2, 0.2, 0.1, 0.2, 0.2, 0.1, 0.2, 0.1, 0.2, 0.0, 0.0, -0.2, 0.0, -0.1, 0.0, -0.2, 0.0, -0.1, 0.0, -0.2, -0.2, 0.0, -0.1, -0.2, -0.2, 0.0, -1.2, -0.2, -0.6, -0.2, -0.2, -0.1, -0.2, -0.1, -0.2, -0.2, -0.1, -0.2, -0.1, -0.2, 0.0, -0.2, 0.0, -0.1, 0.0, -0.2, 0.0, 0.0, -0.2, 0.0, -0.1, 0.0, -0.2, 0.0, 0.0, -0.1, 0.0, -0.2, 0.0, -0.2, 0.0, 0.0, -0.1, 0.0, -0.2, 0.0, -0.1, 0.0, 0.0, -0.2, 0.0, 0.0, 0.2, 0.0, 0.1, 0.0, 0.2, 0.0, 0.0, 0.1, 0.0, 0.2, 0.0, 0.2, 0.0, 0.0, 0.1, 0.0, 0.2, 0.0, 0.1, 0.0, 0.0, 0.2, 0.0, 0.2, 0.0, 0.1, 0.0, 0.0, 0.0, 0.0, -0.1, -0.2, -0.2, -0.1, -0.2, -0.1, -0.2, -0.2, -0.1, -0.2, -0.6, -0.2, -1.3, -0.1, -0.7, -0.1, -1.3, -0.2, -0.6, -0.2, -0.1, -0.2, -0.2, 0.0, 0.2, 0.0, 0.0, 0.0, 0.2, 0.0, 0.0, 0.1, 0.0, 0.0, 0.2, 0.0, 0.0, 0.0, 0.1, 0.0, 0.0, 0.2, 0.0, 0.0, 0.2, 0.0, 0.0, 0.0, 0.1, 0.0, 0.0, 0.2, 0.0, 0.0, 0.1, 0.0, 0.0, -0.1, 0.0, 0.0, -0.2, 0.0, 0.0, -0.1, 0.0, 0.0, -0.2, 0.0, 0.0, 0.0, -0.2, 0.0, 0.0, -0.1, 0.0, 0.0, -0.2, 0.0, 0.0, 0.0, -0.1, 0.0, 0.0, -0.2, 0.0, 0.0, -0.2, 0.0, 0.0, 0.0, -0.1, -0.2, -0.1, -0.2, -0.2, -0.1, -0.2, -0.2, -0.1, -0.2, -0.1, -0.2, -0.2, -0.1, -0.2, -0.1, -0.2, -0.2, -0.1, -0.2, -0.1, -0.2, -1.1, 0.0, -0.7, -0.1, -0.2, -0.2, 0.0, 0.0, 0.2, 0.0, 0.2, 0.0, 0.0, 0.1, 0.0, 0.2, 0.0, 0.0, 0.2, 0.0, 0.1, 0.2, 0.1, 0.2, 0.2, 0.1, 0.2, 0.1, 0.2, 0.2, 0.1, 0.2, 0.1, 0.2, 0.2, 0.1, 0.2, 0.1, 0.2, 0.2, 0.1, 0.2, 0.1, 0.2, 0.0, -0.2, -0.1, -0.2, -0.1, -0.2, -0.2, -0.1, -0.2, -0.1, -0.2, -0.2, -0.1, -0.2, -0.1, -0.2, -0.2, -0.1, -0.2, -0.1, -0.2, -0.2, -0.1, -0.2, -0.1, -0.2, 0.0, -0.2, 0.0, -0.1, -0.2, 0.0, -0.2, 0.0, -0.1, 0.0, -0.2, 0.0, -0.1, -0.2, 0.0, -0.2, 0.0, 0.2, 0.2, 0.0, 0.1, 0.0, 0.2, 0.0, 0.1, 0.0, 0.2, 0.2, 0.0, 0.1, 0.0, 0.2, 0.0, 0.0, -0.2, 0.0, 0.0, -0.1, 0.0, -0.2, 0.0, 0.0, -0.2, 0.0, -0.1, 0.0, 0.0, -0.2, -5.4, -0.2, 0.0, 0.2, 0.1, 0.2, 0.1, 0.2, 0.2, 0.1, 0.2, 0.1, 0.2, 0.2, 0.8, 0.1, 0.7, 0.1, 0.7, 0.0, 0.4, 0.0, 0.0, 0.1, 0.0, 0.1, 0.1, 0.1, 0.0, 0.0, 0.1, 0.0, 0.1, 0.1, 0.0, 0.1, 0.0, 0.1, 0.0, 0.1, 0.1, 0.1, 0.0, 0.1, 0.0, 0.0, 0.1, 0.0, -0.1, 0.0, 0.0, -0.1, 0.0, 0.0, -0.1, -0.1, 0.0, -0.1, 0.0, 0.0, -0.1, 0.0, -0.1, 0.0, -0.1, -0.1, -4.5, 0.0, 0.0, 0.0, 0.1, 0.1, 0.2, 0.0, 0.1, 0.1, 0.1, 0.1, 0.1, 0.1, 0.2, 0.0, 0.1, 0.1, 0.1, 0.1, 0.2, 0.0, 0.2, 0.1, 0.2, 0.2, 0.1, 0.0, 0.2, 0.1, 0.0, 0.6, 0.0, 0.1, 0.0, 0.1, 0.1, 0.1, 0.0, 0.0, 0.1, 0.1, 0.0, 0.1, 0.0, 0.1, 0.0, 0.1, 0.0, 0.1, 0.1, 0.1, 0.0, 0.0, 0.0, 0.0, 0.0, 0.0, -0.1, -0.1, 0.0, -0.1, 0.0, 0.0, -0.1, 0.0, -0.1, -0.1, -3.4, -0.1, 0.0, 0.0, 0.1, 0.1, 0.0, 0.2, 0.0, 0.2, 0.0, 0.1, 0.2, 0.1, 0.0, 0.2, 0.0, 0.2, 0.1, 0.2, 0.2, 0.1, 0.0, 0.5, 0.0, 0.0, 0.2, 0.0, 0.1, 0.0, 0.0, 0.1, 0.1, 0.0, 0.1, 0.0, 0.1, 0.0, 0.1, 0.1, 0.1, 0.0, 0.0, 0.0, 0.0, -0.1, -0.1, 0.0, 0.0, -0.1, -0.1, -2.5, 0.0, 0.0, 0.0, 0.1, 0.0, 0.2, 0.1, 0.0, 0.2, 0.2, 0.1, 0.0, 0.8, 0.0, 0.0, 0.0, 0.1, 0.1, 0.0, 0.1, 0.1, 0.0, 0.1, 0.0, 0.0, 0.0, 0.0, -0.1, -1.5, -0.1, 0.0, 0.1, 0.2, 0.0, 0.1, 0.7, 0.1, 0.0, 0.0, 0.0, 0.0, -0.1, 0.0, -0.1, -0.7, 0.0, -0.2, -0.2, 0.0, -0.1, 0.0, 0.0, 0.0, 1.9, 0.2, 0.0, 0.1, 0.0, 0.1, 0.0, -0.1, 0.0, -0.1, 0.0, -0.1, -0.1, 0.0, 0.0, -0.1, 0.0, -0.1, -0.1, 0.0, -0.1, 0.0, -0.7, 0.0, -0.2, -0.1, -0.1, -0.1, -0.2, 0.0, -0.1, -0.2, 0.0, -0.1, -0.2, 0.0, -0.1, 0.0, 0.0, 0.1, 2.9, 0.2, 0.0, 0.0, 0.1, 0.0, 0.1, 0.0, 0.1, 0.0, 0.0, 0.0, 0.0, -0.1, -0.1, 0.0, -0.1, -0.5, 0.0, -0.1, -0.1, 0.0, -0.1, 0.0, -0.5, 0.0, -0.2, 0.0, -0.1, -0.2, -0.2, -0.1, -0.2, -0.1, -0.1, -0.1, 0.0, -0.2, -0.1, 0.0, -0.2, -0.1, -0.1, -0.1, 0.0, -0.2, -0.1, 0.0, -0.1, 0.0, 0.1, 3.8, 0.2, 0.0, 0.1, 0.0, 0.1, 0.0, 0.1, 0.0, 0.0, 0.1, 0.1, 0.0, 0.1, 0.0, 0.0, 0.1, 0.0, -0.1, 0.0, -0.1, 0.0, -0.1, -0.1, 0.0, -0.1, -0.1, 0.0, -0.1, 0.0, 0.0, -0.1, -0.1, 0.0, -0.1, 0.0, -0.1, -0.1, 0.0, -0.1, -0.1, 0.0, 0.0, -0.4, 0.0, -0.2, -0.2, -0.1, -0.2, 0.0, -0.1, -0.2, -0.2, -0.1, -0.2, 0.0, -0.2, -0.1, -0.2, 0.0, -0.1, 0.0, -0.2, -0.2, 0.0, -0.1, -0.2, 0.0, -0.1, 0.0, -0.2, -0.2, 0.0, -0.1, -0.2, 0.0, 0.0, 0.0, 0.0, 5.0, 0.2, 0.0, 0.0, 0.0, 0.1, 0.0, 0.1, 0.1, 0.0, 0.0, 0.0, 0.1, 0.0, 0.1, 0.1, 0.0, 0.0, 0.1, 0.1, 0.0, 0.0, 0.0, 0.0, 0.0, -0.1, -0.1, 0.0, -0.1, -0.1, 0.0, -0.1, 0.0, -0.1, -0.1, 0.0, -0.1, 0.0, 0.0, -0.1, -0.1, 0.0, -0.1, -0.1, 0.0, -0.1, 0.0, -0.1, -0.1, 0.0, 0.0, 1.5, 0.1, 1.6, 0.2, 0.2, 0.1, 0.2, 0.1, 0.2, 0.2, 0.1, 0.2, 0.1, 0.2, 0.2, 0.1, 0.2, 0.1, 0.2, 0.2, 0.1, 0.2, 0.2, 0.1, 0.2, -0.2, 0.0, -0.1, 0.0, -0.2, 0.0, -0.2, 0.0, -0.1, 0.0, -0.2, 0.0, 0.0, 0.0, 0.2, 0.0, 0.1, 0.0, 0.2, 0.0, 0.2, 0.0, 0.1, 0.0, 0.0, -1.4, 0.0, -0.2, -0.2, -0.1, -0.2, -0.1, -0.2, -0.2, -0.1, -0.2, -0.1, -0.2, -0.2, -0.1, -0.2, -0.1, -0.2, -0.2, -0.1, -0.1, -0.1, -0.1, -0.1, -0.1, -0.1, -0.1, 0.0, -0.1, -0.1, -0.1, -0.2, 0.0, -0.1, -0.1, -0.1, 0.0, 1.0, 0.2, 0.1, 1.3, 0.2, 0.1, 0.2, 0.1, 0.2, 0.2, 0.1, 0.2, 0.1, 0.2, 0.2, 0.1, 0.2, 0.1, 0.2, -0.1, -0.1, 0.0, -0.1, -0.1, -0.1, -0.1, 0.0, 0.0, 0.0, 0.0, 0.0, 0.0, 0.0, 0.1, 0.1, 0.1, 0.1, 0.0, -1.4, 0.0, -0.1, -0.1, -0.1, -0.2, -0.1, -0.1, -0.1, -0.2, -0.1, -0.2, -0.1, 0.0, -0.1, -0.1, -0.1, -0.1, 0.0, 0.0, -0.1, 0.0, -0.1, -0.1, 0.0, -0.1, 0.0, 0.0, -0.1, -0.1, -0.1, -0.1, 0.0, 0.0, 0.5, 0.2, 0.0, 0.1, 0.1, 0.1, 1.0, 0.1, 0.2, 0.1, 0.0, 0.2, 0.2, 0.1, 0.0, 0.2, 0.1, 0.1, -0.1, 0.0, 0.0, -0.1, 0.0, -0.1, 0.0, -0.1, 0.0, 0.0, 0.0, 0.0, 0.0, 0.1, 0.0, 0.0, -1.2, 0.0, -0.2, -0.1, -0.2, -0.1, 0.0, -0.1, -0.1, -0.1, -0.1, 0.0, 0.0, 0.1, 0.1, 0.1, 0.1, 0.1, 0.1, 0.1, 0.6, 0.2, 0.1, -0.1, 0.0, 0.0, 0.0, 0.0, 0.0, 0.0, 0.0, -0.3, 0.0, -0.2, -0.1, -0.1, -0.1, -0.2, -0.1, 0.1, 0.0, 0.1, 0.0, 1.2, 0.0, 0.0, 0.0, 0.0, 0.0, 0.0, 0.0, 0.0, 0.1, 0.0, 0.1, 0.0, 0.0, 0.0, -0.2, -0.2, 0.0, -0.1, -0.2, -0.1, -0.8, 0.0, -0.2, 0.0, -0.2, 0.0, -0.1, -0.1, -0.1, -0.1, 0.0, 0.1, 0.0, 0.1, 0.1, 0.0, 0.1, 0.0, 0.1, 0.1, 0.0, 0.0, 0.1, 0.1, 0.1, 0.2, 0.1, 0.2, 0.0, 0.2, 0.1, 0.0, 1.4, 0.0, -0.1, 0.0, 0.0, -0.1, 0.0, -0.1, 0.0, 0.0, 0.0, 0.1, 0.0, 0.1, 0.0, 0.0, 0.1, 0.1, 0.0, 0.1, 0.0, 0.1, -0.1, -0.1, -0.2, 0.0, -0.2, -0.1, -0.1, -0.1, -0.1, -0.2, -0.1, -0.1, -0.1, -0.2, -0.1, 0.0, -0.1, -1.1, -0.1, -0.1, -0.1, -0.1, -0.1, -0.6, -0.1, 0.1, 0.0, 0.1, 0.1, 0.0, 0.1, 0.0, 0.1, 0.1, 0.0, 0.0, 0.1, 0.1, 0.0, 0.1, 0.0, 0.1, 0.1, 0.0, 0.1, 0.0, 0.1, 0.1, 0.2, 0.1, 0.2, 0.1, 0.2, 0.2, 0.1, 0.2, 0.1, 0.2, 0.2, 0.1, 0.2, 0.0, 1.3, 0.0, 0.0, -0.1, -0.1, 0.0, 0.0, -0.1, -0.1, 0.0, -0.1, 0.0, 0.0, 0.0, 0.0, 0.0, 0.1, 0.0, 0.1, 0.1, 0.0, 0.0, 0.1, 0.1, 0.0, 0.1, 0.0, 0.1, 0.1, -0.2, -0.1, -0.2, -0.2, 0.0, -0.1, -0.2, -0.1, -0.2, -0.2, -0.1, -0.2, -0.1, -0.2, -0.2, -0.1, -0.2, -0.1, -0.2, -1.4, -0.2, -0.1, -0.1, -1.2, 0.1, 0.0, 0.0, 0.1, 0.1, 0.0, 0.1, 0.0, 0.1, 0.1, 0.0, 0.1, 0.0, 0.1, 0.1, 0.0, 0.0, 0.1, 0.1, 0.0, 0.1, 0.0, 0.1, 0.1, 0.0, 0.1, 0.1, 0.0, 0.1, 0.0, 0.1, 0.1, 0.1, 0.2, 0.2, 0.1, 0.2, 0.1, 0.2, 0.2, 0.1, 0.2, 0.1, 0.2, 0.2, 0.1, 0.2, 0.1, 0.2, 0.2, 0.1, 0.2, 0.1, 0.9, 0.1, 0.2, 0.1, 0.2, 0.0, 0.2, 0.0, 0.1, 0.0, 0.2, 0.1, 0.2, 0.0, -0.3, 0.0, -0.1, -0.1, 0.0, -0.1, 0.0, 0.0, 0.0, -0.1, -0.1, 0.0, -0.1, 0.0, -0.1, -0.1, 0.0, 0.0, 0.0, -0.1, -0.1, 0.0, -0.1, 0.0, 0.0, -0.1, -0.1, 0.0, -0.2, -0.1, -0.2, -0.2, -0.1, -0.2, -0.1, -0.2, -0.2, -0.1, -0.2, -0.1, -0.2, -0.2, -0.1, -0.2, -0.8, -0.1, 0.0, -0.7, -0.1, 0.1, 0.0, 0.1, 0.1, 0.1, 0.0, 0.0, 0.1, 0.1, 0.2, 0.1, 0.2, 0.1, 0.2, 0.2, 0.1, 0.2, 0.1, 0.2, 0.2, 0.1, 0.2, 0.1, 0.2, 0.2, 0.1, 0.2, 0.1, 0.2, 0.2, 0.1, 0.2, 0.2, 0.1, 0.1, 0.1, 0.0, 0.1, 0.2, 0.0, -0.4, 0.0, -0.1, 0.0, 0.0, 0.0, -0.1, 0.0, 0.0, -0.1, 0.0, -0.1, 0.0, 0.0, -0.1, 0.0, -0.1, 0.0, 0.0, 0.0, -0.1, 0.0, 0.0, -0.2, -0.1, -0.1, -0.1, -0.1, -0.1, -0.1, 0.0, -0.2, -0.1, -0.1, -0.1, -0.1, -0.1, 0.0, -0.1, -0.2, 0.0, -0.2, -0.5, -0.1, 0.0, -0.1, -0.1, 0.0, -0.3, -0.1, 0.0, 0.1, 0.0, 0.1, 0.0, 0.1, 0.1, 0.2, 0.1, 0.1, 0.1, 0.2, 0.1, 0.1, 0.1, 0.2, 0.1, 0.2, 0.1, 0.0, 0.2, 0.2, 0.1, 0.1, 0.1, 0.1, 0.2, 0.1, 0.1, 0.1, 0.2, 0.0, 0.1, 0.1, 0.0, -0.5, 0.0, 0.0, -0.1, 0.0, -0.1, -0.1, 0.0, -0.1, 0.0, -0.1, 0.0, -0.2, -0.1, -0.1, -0.1, -0.1, -0.1, -0.1, 0.0, -0.2, -0.1, 0.0, -0.1, -0.1, -0.1, -0.1, 0.0, -0.1, 0.0, -0.1, -0.1, -0.1, 0.0, 0.1, 0.2, 0.1, 0.2, 0.2, 0.1, 0.2, 0.1, 0.2, 0.2, 0.1, 0.2, 0.0, -0.8, 0.0, 0.3, -0.1, -0.1, -0.1, -0.2, -0.1, -0.1, -0.1, 0.0, 0.0, 0.0, 0.2, 0.0, 0.1, 0.1, 0.1, 0.1, 0.0, 0.2, 0.2, 0.0, 0.1, 0.1, 0.0, 0.1, 0.0, 0.0, 0.1, 0.0, 0.0, 0.4, 0.0, 0.0, -0.1, -0.1, -0.2, -0.1, -0.1, -0.1, -0.1, -0.2, -0.2, 0.0, -0.1, -0.2, -0.1, -0.2, 0.0, -0.2, -0.1, -0.2, -0.1, -0.1, -0.1, -0.1, -0.1, 0.0, 0.0, 0.0, 0.1, 0.1, 0.1, 0.1, 0.0, 0.1, 0.0, 0.1, 0.4, 0.1, 0.1, 0.1, 0.1, 0.1, 0.1, 0.0, 0.2, 0.0, 0.2, 0.1, 0.0, 0.2, 0.0, 0.1, 0.2, 0.0, 0.0, 0.0, 0.1, 0.0, 0.1, 0.0, 0.0, 0.1, 0.0, 0.1, 0.0, 0.1, 0.0, 0.0, 0.0, 0.1, 0.0, 0.3, 0.0, -0.1, 0.0, -0.1, 0.0, -0.2, -0.2, -0.1, -0.2, -0.2, -0.1, -0.2, 0.0, -0.1, -0.2, -0.2, -0.1, -0.2, -0.1, -0.2, -0.2, -0.1, -0.2, -0.1, -0.2, -0.2, -0.1, -0.2, 0.0, -0.1, -0.1, 0.0, -0.1, 0.0, 0.0, -0.1, -0.1, 0.0, 0.0, 0.5, 0.1, 0.1, 0.0, 0.1, 0.0, 0.7, 0.1, 0.1, 0.1, 0.1, 0.1, 0.1, 0.0, 0.2, 0.1, 0.0, 0.2, 0.1, 0.1, 0.1, 0.0, 0.2, 0.1, 0.0, 0.2, 0.1, 0.1, 0.1, 0.0, 0.1, 0.0, 0.1, 0.0, 0.0, 0.1, 0.1, 0.0, 0.0, 0.1, 0.0, 0.0, 0.1, 0.0, 0.1, 0.0, 0.0, 0.1, 0.0, 0.0, 0.1, 0.0, 0.1, 0.0, 0.0, 0.3, -0.2, -0.1, 0.0, 0.0, -0.1, -0.1, 0.0, -0.1, 0.0, -0.2, -0.1, -0.2, -0.2, -0.1, -0.2, -0.2, -0.1, -0.2, -0.1, -0.2, -0.2, -0.1, -0.2, -0.1, -0.2, -0.2, -0.1, -0.2, -0.1, -0.2, -0.2, -0.1, -0.2, -0.1, -0.2, -0.2, -0.1, -0.1, -0.1, 0.0, 0.0, -0.1, 0.0, -0.1, -0.1, 0.0, 0.0, -0.1, -0.1, 0.0, 0.0, 0.2, 0.2, 0.5, 0.1, 0.0, 0.0, 0.4, 0.6, 0.0, 0.1, 0.2, 0.3, 0.1, 0.1, 0.1, 0.1, 0.1, 0.1, 0.1, 0.1, 0.1, 0.1, 0.1, 0.1, 0.1, 0.1, 0.1, 0.1, 0.2, 0.1, 0.0, 0.2, 0.2, 0.1, 0.0, 0.0, 0.1, 0.1, 0.0, 0.1, 0.0, 0.1, 0.1, 0.0, 0.0, 0.0, 0.1, 0.1, 0.0, 0.1, 0.0, 0.0, 0.1, 0.1, 0.0, 0.0, 0.1, 0.0, 0.1, 0.1, 0.0, 0.0, 0.1, 0.5, 0.2, 0.2, 2.5, 0.0, 0.4, 0.0, 0.0, 0.0, 0.1, 0.1, 0.1, 0.0, 0.1, 0.1, 0.0, 0.1, 0.1, 0.1, 0.0, 0.1, 0.0, 0.1, 0.1, 0.1, 0.0, 0.1, 0.1, 0.0, 0.1, 0.1, 0.0, 0.1, 0.0, -0.1, -0.2, -0.2, -0.1, -0.2, -0.1, -0.2, -0.2, -0.1, -0.2, -0.1, -0.2, -1.0, -0.1, -0.2, -0.2, -0.1, -0.2, -0.1, -1.0, -0.2, -0.1, -0.2, -0.1, -0.2, -0.2, 0.1, 0.1, 0.0, 0.1, 0.0, 0.1, 0.1, 0.0, 0.0, 0.0, 0.1, 0.1, 0.0, 0.1, 0.0, 0.0, 0.1, 0.1, 0.0, 0.0, 0.1, 0.0, 0.1, 0.1, 0.0, 0.0, 0.1, 0.1, 0.0, 0.0, 0.1, 0.0, 1.3, 0.0, 0.7, 0.0, 0.0, 0.1, 0.0, 0.0, 0.1, 0.1, 0.0, 0.0, 0.1, 0.0, 0.1, 0.0, 0.1, 0.0, 0.1, 0.1, 0.0, 0.0, 0.1, 0.0, 0.0, 0.1, 0.1, 0.0, 0.1, 0.1, 0.0, 0.0, 0.0, 0.0, 0.0, -0.2, -0.2, -0.1, -0.2, -0.1, -0.2, -0.2, -0.1, -0.7, -0.1, -0.2, -0.2, -0.1, -0.2, -0.1, -0.7, -0.1, -0.2, -0.1, 0.1, 0.0, 0.0, 0.1, 0.0, 0.1, 0.0, 0.0, 0.0, 0.1, 0.0, 0.0, 0.1, 0.0, 0.1, 0.0, 0.1, 0.0, 0.0, 0.0, 0.1, 0.0, 0.1, 0.0, 0.0, 0.1, 0.0, 0.1, 0.0, 0.0, 0.1, 0.0, 0.2, 0.1, 0.0, 0.8, 0.0, 0.1, 0.0, 0.1, 0.0, 0.1, 0.1, 0.1, 0.0, 0.1, 0.0, 0.1, 0.1, 0.1, 0.0, -0.2, -0.2, -0.1, -0.7, -0.1, -0.2, -0.2, -0.1, -0.2, -0.1, -0.2, 0.0, 0.0, 0.1, 0.0, 0.1, 0.0, 0.1, 0.0, 0.1, 0.0, 0.1, 0.0, 0.0, 0.1, 0.0, 0.4, 0.0, 0.1, 0.1, 0.1, 0.0, -0.2, -0.1, -0.2, 0.0, 0.0, 0.1, 0.0, 0.1, -0.2, -0.1, 0.0, -0.1, 0.0, 0.0, -0.1, 0.0, -0.1, 0.0, 0.0, 0.1, 0.1, 0.2, 0.2, 0.1, 0.2, 0.2, 0.1, 0.2, 0.0, -0.1, 0.0, -0.1, 0.0, -0.1, 0.0, -0.1, -0.1, 0.0, 0.0, 0.0, -0.8, 0.0, 0.0, 0.0, -0.1, 0.0, -0.1, 0.0, 0.0, -0.1, 0.0, 0.0, -0.1, 0.0, -0.1, 0.0, 0.0, -0.1, 0.0, -0.1, 0.0, 0.0, -0.1, 0.0, 0.0, 0.0, -0.1, 0.0, 0.1, 0.1, 0.2, 0.2, 0.1, 0.2, 0.1, 0.2, 0.2, 0.1, 0.7, 0.1, 0.2, 0.2, 0.1, 0.2, 0.1, 0.0, -0.1, 0.0, -0.1, 0.0, -0.1, 0.0, -0.1, 0.0, 0.0, -0.1, -0.1, 0.0, 0.0, -0.1, -0.1, 0.0, -0.1, 0.0, 0.0, -0.1, -0.1, 0.0, 0.0, 0.0, -0.5, -0.9, -0.2, 0.0, 0.0, -0.1, -0.1, 0.0, 0.0, -0.1, 0.0, 0.0, -0.1, 0.0, -0.1, 0.0, 0.0, -0.1, 0.0, 0.0, -0.1, 0.0, -0.1, 0.0, 0.0, -0.1, -0.1, 0.0, 0.0, -0.1, 0.0, 0.0, -0.1, 0.0, -0.1, 0.0, 0.0, 0.2, 0.1, 0.2, 0.2, 0.8, 0.1, 0.2, 0.1, 0.2, 0.2, 0.1, 0.8, 0.2, 0.2, 0.1, 0.2, 0.1, 0.2, 0.2, 0.1, 0.1, 0.1, 0.1, 0.1, 0.0, -0.1, 0.0, -0.1, 0.0, 0.0, -0.1, 0.0, -0.1, 0.0, -0.1, 0.0, -0.1, -0.1, 0.0, 0.0, -0.1, 0.0, -0.1, 0.0, -0.1, 0.0, -0.1, 0.0, -0.1, 0.0, 0.0, -0.1, 0.0, -0.1, -0.1, 0.0, -0.1, 0.0, -0.5, -1.8, -0.2, 0.0, -0.1, 0.0, 0.0, -0.1, -0.1, 0.0, 0.0, -0.1, -0.1, 0.0, -0.1, 0.0, 0.0, 0.0, -0.1, -0.1, 0.0, -0.1, 0.0, -0.1, -0.1, 0.0, 0.0, 0.0, -0.1, -0.1, 0.0, -0.1, 0.0, -0.1, 0.0, -0.1, 0.0, 0.0, 0.2, 0.1, 0.2, 0.2, 0.1, 0.2, 0.1, 0.2, 1.0, 0.1, 0.2, 0.1, 0.2, 0.2, 0.1, 1.0, 0.2, 0.1, 0.2, 0.1, 0.2, 0.2, 0.1, 0.2, 0.1, 0.2, 0.2, 0.1, 0.2, 0.1, 0.2, 0.0, -0.1, -0.1, 0.0, -0.1, 0.0, 0.0, -0.1, -0.1, 0.0, -0.1, 0.0, -0.1, -0.1, 0.0, 0.0, -0.1, -0.1, 0.0, -0.1, 0.0, -0.1, 0.0, -0.1, 0.0, -0.1, 0.0, -0.1, -0.1, 0.0, 0.0, -0.1, -0.1, 0.0, -0.1, 0.0, -0.1, 0.1, 0.0, 0.1, 0.2, 0.2, 0.1, 0.2, 0.0, 0.1, 0.0, 0.2, 0.0, 0.2, 0.0, 0.1, 0.0, 1.3, 0.0, 0.2, 0.1, 0.2, 0.2, 0.1, 0.2, 0.1, 0.2, 0.2, 0.1, 0.2, 0.1, 0.2, 0.2, 0.1, 0.2, 0.1, 0.2, 0.2, 0.1, 0.2, 0.1, 0.2, 0.2, 0.1, 0.1, 0.0, -0.1, -0.1, 0.0, -0.1, -0.1, -0.2, 0.0, -0.1, -0.2, -0.1, -0.1, -0.1, -1.0, -0.1, -0.2, -0.1, -0.2, -0.2, -0.1, -0.2, -0.1, -0.2, -0.2, -0.1, -0.1, -0.1, -0.1, 0.0, -0.1, 0.0, -0.1, -0.1, -0.1, 0.0, -0.1, 0.0, -0.1, -0.1, -0.1, -0.1, 0.0, -0.1, 0.0, -0.1, -0.1, 0.0, -0.1, -0.1, -0.1, 0.0, -0.1, -0.1, 0.2, 0.2, 0.1, 0.0, 0.1, 0.1, 0.1, 0.0, 1.3, 0.0, 0.0, 0.2, 0.1, 0.1, 0.1, 0.2, 0.1, 0.0, 0.2, 0.1, 0.1, 0.1, 0.2, 0.1, 0.0, 0.2, 0.1, 0.1, 0.1, 0.2, 0.1, 0.0, 0.2, 0.1, 0.1, 0.1, -0.1, 0.0, 0.0, -0.1, -0.1, 0.0, -0.1, -0.1, -0.1, 0.0, -0.1, -0.1, 0.0, -0.1, -0.7, -0.1, -0.1, -0.1, -0.1, -0.1, -0.3, -0.1, -0.1, -0.1, -0.1, -0.1, 0.0, 0.0, -0.1, 0.0, -0.1, -0.1, 0.0, 0.0, -0.1, 0.0, 0.0, -0.1, -0.1, 0.0, -0.1, -0.1, 0.0, 0.0, -0.1, 0.0, 0.0, -0.1, -0.1, 0.0, -0.1, 0.0, -0.1, 0.0, 0.0, 0.1, 0.1, 0.0, 0.1, 0.0, 1.4, 0.0, 0.1, 0.2, 0.1, 0.2, 0.2, 0.1, 0.2, 0.1, 0.2, 0.1, 0.0, -0.1, 0.0, -0.2, 0.0, 0.0, -0.1, -0.1, -0.3, -0.1, -0.1, -0.1, -0.1, 0.0, -0.2, -0.1, -0.1, 0.0, -0.1, -0.1, -0.1, 0.0, -0.1, -0.1, 0.0, -0.1, -0.1, 0.0, 0.9, 0.0, 0.2, 0.1, 0.1, 0.0, -0.1, 0.0, -0.1, -0.1, -0.4, 0.0, 0.0, 0.1, 0.1, 0.0, 0.1, 0.0, 0.2, 0.1, 0.4, 0.1, 0.0, 0.1, 0.0, 0.0, -0.1, -0.1, -0.2, -0.1, -0.1, -0.1, -0.1, 0.0, -1.5, 0.0, 0.0, 0.1, 0.0, 0.1, 0.1, 0.0, 0.0, 0.1, 0.0, 0.1, 0.0, 0.1, 0.0, 0.1, 0.0, 0.1, 0.0, 0.1, 0.0, 0.0, 0.1, 0.1, 0.0, 0.1, 0.1, 0.0, 0.1, 0.1, 0.1, 0.1, 0.0, 0.2, 0.1, 0.1, 0.5, 0.1, 0.0, 0.1, 0.1, 0.0, 0.1, 0.1, 0.1, 0.0, 0.0, 0.1, 0.0, -0.1, -0.2, -0.1, -0.1, -0.1, -0.2, 0.0, -0.1, -0.2, -0.1, -0.1, -0.1, -0.2, -0.1, 0.0, -0.2, -0.1, -0.1, -0.1, 0.0, -1.4, 0.0, -0.1, 0.0, -0.1, 0.0, -0.1, -0.1, 0.0, 0.0, 0.0, 0.0, 0.1, 0.0, 0.1, 0.0, 0.1, 0.0, 0.1, 0.1, 0.0, 0.0, 0.1, 0.0, 0.1, 0.0, 0.1, 0.0, 0.1, 0.0, 0.1, 0.0, 0.0, 0.1, 0.1, 0.0, 0.1, 0.0, 0.1, 0.0, 0.1, 0.0, 0.1, 0.0, 0.1, 0.1, 0.2, 0.0, 0.1, 0.2, 0.3, 0.2, 0.0, 0.1, 0.2, 0.0, 0.8, 0.0, 0.1, 0.0, 0.1, 0.1, 0.0, 0.2, 0.0, 0.1, 0.0, 0.1, 0.1, 0.0, 0.1, 0.0, 0.1, 0.0, 0.1, -0.2, 0.0, -0.1, -0.2, -0.1, 0.0, -0.2, -0.1, -0.1, -0.1, -0.2, -0.1, 0.0, -0.2, -0.1, -0.1, -0.1, -0.2, -0.1, 0.0, -0.2, -0.1, -0.1, -0.1, -0.2, -0.1, 0.0, -0.2, -0.1, -0.1, -0.1, 0.0, -1.4, 0.0, -0.1, 0.0, -0.1, 0.0, -0.1, -0.1, 0.0, 0.0, -0.1, -0.1, -0.1, 0.0, -0.2, -0.1, 0.1, 0.0, 0.1, 0.1, 0.0, 0.0, 0.1, 0.0, 0.1, 0.1, 0.0, 0.0, 0.1, 0.1, 0.0, 0.1, 0.0, 0.1, 0.1, 0.0, 0.0, 0.1, 0.0, 0.1, 0.1, 0.0, 0.0, 0.1, 0.1, 0.0, 0.1, 0.0, 0.1, 0.1, 0.0, 0.0, 0.1, 0.1, 0.0, 0.1, 0.0, 0.1, 0.1, 0.1, 0.1, 0.1, 0.1, 0.1, 0.1, 0.1, 0.1, 0.1, 0.1, 0.1, 0.5, 0.1, 0.1, 0.1, 1.1, 0.0, 0.1, 0.1, 0.3, 0.0, 0.0, 0.1, 0.1, 0.1, 0.0, 0.1, 0.1, 0.0, 0.0, 0.1, 0.1, 0.0, 0.1, 0.0, 0.0, 0.0, 0.0, -0.1, 0.0, -0.2, -0.2, -0.1, -0.2, -0.1, -0.1, -0.1, -0.1, -0.1, -0.1, -0.2, -0.2, -0.1, -0.1, -0.1, -0.1, -0.2, -0.2, -0.1, -0.1, -0.1, -0.1, -0.2, -0.2, -0.1, -0.1, -0.1, -0.1, -0.1, -0.1, -0.2, -0.1, -0.2, -0.1, -0.7, 0.0, -0.2, 0.2, 0.0, 0.2, 0.0, 0.1, 0.0, 0.2, 0.0, 0.0, 0.0, -0.2, 0.0, 0.0, 1.3, 0.0, 0.2, 0.1, 0.2, 0.2, 0.1, 0.2, 0.1, 0.2, 0.2, 0.1, 0.2, 0.1, 0.2, 0.2, 0.1, 0.2, 0.1, 0.2, 0.2, 0.1, 0.2, 0.2, 0.1, 0.2, 0.1, 0.1, 0.1, 0.0, 0.0, 0.1, 0.1, 0.0, 0.0, 0.0, 0.0, 0.1, 0.0, -0.1, 0.0, 0.0, 0.0, 0.0, 0.0, -0.1, -0.1, 0.0, 0.0, 0.0, -0.1, 0.0, -0.1, -0.1, -0.2, -0.1, -0.2, -0.2, -0.1, -0.2, -0.2, -0.1, -0.2, -0.1, -0.2, -0.2, -0.1, -0.2, -0.1, -0.2, -0.2, -0.1, -0.2, -0.1, -0.2, -0.2, -0.1, -0.2, -0.1, -0.2, -0.2, -0.1, -0.2, 0.1, 0.1, 0.1, 0.0, 0.0, 0.0, 0.0, 0.0, 0.0, 1.3, 0.3, 0.2, 0.0, 0.2, 0.1, 0.2, 0.0, 0.1, 0.2, 0.0, 0.2, 0.1, 0.2, 0.0, 0.1, 0.2, 0.2, 0.0, 0.1, 0.2, 0.2, 0.1, 0.0, 0.0, 0.1, 0.0, 0.1, 0.0, 0.0, 0.0, -0.1, 0.0, -0.1, 0.0, 0.0, 0.0, -0.1, 0.0, 0.0, 0.0, -0.2, -0.2, -0.1, 0.0, -0.2, -0.2, -0.1, 0.0, -0.2, -0.1, 0.0, -0.2, -0.2, -0.1, 0.0, -0.2, -0.1, 0.0, -0.2, -0.2, -0.1, 0.0, -0.2, -0.1, 0.0, -0.2, -0.1, -0.1, -0.1, -0.1, 0.0, 0.1, 0.0, 0.0, 1.3, 0.0, 0.1, 0.2, 0.1, 0.2, 0.2, 0.1, 0.2, 0.1, 0.2, 0.2, 0.1, 0.0, 0.0, 0.0, -0.1, 0.0, 0.0, 0.0, 0.0, -0.2, -0.2, -0.1, -0.2, -0.1, -0.2, -0.2, -0.1, -0.2, -0.1, -0.2, 0.0, 0.8, 0.0, 0.2, 0.1, 0.2, 0.0, -0.2, -0.1, -0.4, 0.1, 0.1, 0.2, 0.1, 0.1, 0.1, 0.1, 0.1, 0.0, 0.1, 0.0, 0.0, -0.2, -0.1, -0.2, -0.1, 0.0, -0.2, -0.1, -0.1, 0.0, -1.4, 0.0, 0.0, 0.0, 0.2, 0.0, 0.1, 0.2, 0.1, 0.0, 0.2, 0.2, 0.1, 0.0, 0.2, 0.1, 0.0, 0.2, 0.2, 0.1, 0.0, 0.2, 0.1, 0.0, 0.2, 0.2, 0.1, 0.0, 0.1, 0.1, 0.0, 0.0, 0.0, 0.0, 0.1, 0.0, 0.1, 0.0, -0.1, 0.0, -0.1, 0.0, 0.0, -0.2, 0.0, -0.1, -0.2, -0.2, 0.0, -0.1, -0.2, -0.1, -0.1, -0.1, -0.2, 0.0, -0.1, -0.2, -0.1, -0.1, -0.1, -0.2, 0.0, -1.2, 0.0, 0.0, 0.0, -0.1, 0.0, -0.1, 0.0, 0.0, 0.0, 0.1, 0.1, 0.1, 0.2, 0.1, 0.0, 0.2, 0.1, 0.1, 0.1, 0.1, 0.1, 0.1, 0.2, 0.1, 0.1, 0.1, 0.2, 0.0, 0.1, 0.2, 0.1, 0.1, 0.1];

    ! Set speed in mm/s and corner rounding.
    VAR speeddata mySpeed:=v500;
    VAR zonedata myZone:=z10;

    ! Set home point.
    CONST robtarget pHome:=[[-774.08,-2214.17,1285.95],[0.000170095,0.000237984,0.707577,-0.706636],[-2,0,-2,1],[9E+09,9E+09,9E+09,9E+09,9E+09,9E+09]];

    ! Set initial point.
    VAR robtarget pCurrent:=[[-774.08,-2214.17,1285.95],[0.000170093,0.000237981,0.707577,-0.706636],[-2,0,-2,1],[9E+09,9E+09,9E+09,9E+09,9E+09,9E+09]];

    PROC mane()
          MoveL pHome,mySpeed,myZone,tspray\WObj:=wobj0;
          MoveL pCurrent,mySpeed,myZone,tspray\WObj:=wobj0;

        FOR i FROM 2 TO 5 DO
            pCurrent.trans:=[
                pCurrent.trans.x+x_coords_rel{i},
                pCurrent.trans.y+y_coords_rel{i},
                pCurrent.trans.z+z_coords_rel{i}
            ];
            MoveL pCurrent,mySpeed,myZone,tspray\WObj:=wobj0;
        ENDFOR
    ENDPROC
ENDMODULE
